// SIMATIC STEP 7 (V5.x) project PLC_PRV
// CPU: CPU 317-2 PN/DP
// station: Hardware
// station: SIMATIC 300 Station
// station: P_ADR_BUS
// program: S7 Program(6)

SYMBOL_TABLE
"RS485_chenal1"	DB 71	FB 72
"RS485_chanel2"	DB 72	FB 72
"RS485_chanel3"	DB 73	FB 72
"RS485_chanel4"	DB 74	FB 72
"KerVal1"	DB 101	FB 1
"ValGluchPerf"	DB 102	FB 1
"VidsmokVal"	DB 103	FB 1
"CalcRPM_Setka"	DB 104	FB 1
"CalcRPM_Gauch"	DB 105	FB 1
"CalcRPM_KerVal2"	DB 106	FB 1
"CalcRPM_JolVal"	DB 107	FB 1
"CalcRPM_Sushka1"	DB 108	FB 1
"CalcRPM_Sushka2"	DB 109	FB 1
"CalcRPM_Sushka3"	DB 110	FB 1
"CalcRPM_Sushka4"	DB 111	FB 1
"CalcRPM_KlejPresBNV1"	DB 112	FB 1
"CalcRPM_KlejPresBNV2"	DB 113	FB 1
"CalcRPM_KlejPresBNV3"	DB 114	FB 1
"CalcRPM_KlejPresBNV4"	DB 115	FB 1
"CalcRPM_KlejPresRuhVal"	DB 116	FB 1
"CalcRPM_KlejPresNeRuhVal"	DB 117	FB 1
"CalcRPM_Sushka5"	DB 118	FB 1
"CalcRPM_Sushka6"	DB 119	FB 1
"CalcRPM_Sushka7"	DB 120	FB 1
"CalcRPM_Kalandr"	DB 121	FB 1
"CalcRPM_Nakat"	DB 122	FB 1
"PaperVed1"	DB 123	FB 1
"PaperVedVal2"	DB 124	FB 1
"CalcRPM_PapVedVal3"	DB 125	FB 1
"CalcRPM_RozgonTambur"	DB 126	FB 1
"SpeedCalc_KombiPress"	DB 130	FB 2
"SpeedCalc_Sitka"	DB 131	FB 2
"CalcSpeed_Pres3"	DB 132	FB 2
"CalcSpeed_Sushka1"	DB 133	FB 2
"CalcSpeed_Sushka2"	DB 134	FB 2
"CalcSpeed_Sushka3"	DB 135	FB 2
"CalcSpeed_Sushka4"	DB 136	FB 2
"CalcSpeed_KlejPress"	DB 137	FB 2
"CalcSpeed_Sushka5"	DB 138	FB 2
"CalcSpeed_Sushka6"	DB 139	FB 2
"CalcSpeed_Sushka7"	DB 140	FB 2
"Signals_To_Nakat"	DB 201	DB 201
"PapVed1_Speed_Unit"	DB 203	FB 2
"PapVed2_Speed_Unit"	DB 204	FB 2
"PapVed3_Speed_Unit"	DB 205	FB 2
"Calc_RPM_Privod"	FB 1	FB 1	// Rozrahunok_RPM_privodiv
"Calc_Speed_Unit"	FB 2	FB 2	// Rozrahunok_shvidkosti_uzlov
"SEND"	FB 60	FB 60
"RECEIVE"	FB 61	FB 61
"RTU_MB_MASTER"	FB 72	FB 72
"RS485_1"	FC 1	FC 1	// RS485_1_Chanel
"RS485_2"	FC 2	FC 2	// RS485_2_chanel
"RS485_Runchanel3"	FC 3	FC 3
"RS485_RunChanel4"	FC 4	FC 4
"Speed_Calculation"	FC 10	FC 10	// Speed_Calculation
"RPM_Calculation"	FC 11	FC 11	// RPM_Calculation
"Speed_Intens"	FC 12	FC 12
"Calc_RPM_to_Hz"	FC 14	FC 14
"Calc_Zaprav_Speed"	FC 15	FC 15
"Check_AlarmPPS"	FC 30	FC 30
"UNSCALE"	FC 106	FC 106	// Unscaling Values
"SER_CFG"	FC 216	FC 216
"Kn_Zap_vidsm_val"	I 0.0	BOOL
"Vidsm_val_kontr_vkl"	I 0.2	BOOL
"Vidsm_val_kontR_blok"	I 0.4	BOOL
"Jolob_val_kont_kn_zapob"	I 0.5	BOOL
"Jolob_val_kont_vkl"	I 0.7	BOOL
"Jolob_val_kont_blok"	I 1.0	BOOL
"Keram_val1_kont_kn_zapob"	I 1.1	BOOL
"Keram_val1_kont_vkl"	I 1.3	BOOL
"Keram_val_1_kont_blok"	I 1.5	BOOL
"Ker_val2_konT_blok"	I 2.1	BOOL
"Ker_val_2_kont_kn_zapob"	I 2.4	BOOL
"Ker_val_2_kont_vkl"	I 2.6	BOOL
"Gluh_perf_kontr_kn_zapob"	I 3.0	BOOL
"Kalandr_kontrol_kn_zap"	I 9.0	BOOL
"Kalandr_kont_vkl"	I 9.2	BOOL
"Kalandr_kont_blokuvan"	I 9.4	BOOL
"Rozg_Tamb_Kn_Zap"	I 9.5	BOOL
"Rozg_Tamb_Kont_Vkl"	I 9.7	BOOL
"Rozg_Tamb_Kont_blok"	I 10.0	BOOL
"Nakat_kontrol_kn_zapob"	I 10.1	BOOL
"Nakat_kontrol_vkl"	I 10.3	BOOL
"Nakat_kontrol_blok"	I 10.5	BOOL
"MST_Zab_Zap_pres1_2_pik"	I 12.3	BOOL
"Z_MST_ZAB_zap_3_presu"	I 12.5	BOOL
"rez"	I 12.6	BOOL
"En_SitkVrusi"	M 20.0	BOOL	// Імітація сигналу на SCADA
"En_KombPresVroboti"	M 20.2	BOOL	// Імітація сигналу на SCADA
"Suska3_cor-"	M 20.3	BOOL
"En_Pres3Vroboti"	M 20.4	BOOL	// Імітація сигналу на SCADA
"Suska3_Pidtagnut"	M 20.5	BOOL
"Pusk_3pres"	M 20.6	BOOL	// Включити 3й прес HMI
"SitkaGaush_pusk"	M 20.7	BOOL	// Включити Сітка + гауч HMI_51
"Serv_mode_Sitka_Gauch"	M 21.1	BOOL
"Serv_mode_Kombi_Pres"	M 21.2	BOOL
"Serv_mode_Pres_3"	M 21.3	BOOL
"Serv_mode_Suska1"	M 21.6	BOOL
"Serv_mode_Suska2"	M 21.7	BOOL
"Serv_mode_Suska3"	M 22.0	BOOL
"Serv_mode_Suska4"	M 22.1	BOOL
"Serv_mode_BumNapr1"	M 22.2	BOOL
"Serv_mode_BumNapr2"	M 22.3	BOOL
"Serv_mode_BumNapr3"	M 22.4	BOOL
"Serv_mode_BumNapr4"	M 22.5	BOOL
"Serv_mode_RuhVal"	M 22.6	BOOL
"Serv_mode_NeruhVal"	M 22.7	BOOL
"Serv_mode_Suska5"	M 23.0	BOOL
"Serv_mode_Suska6"	M 23.1	BOOL
"Serv_mode_Suska7"	M 23.2	BOOL
"Serv_mode_PapVed3"	M 23.3	BOOL
"Serv_mode_Kalandr"	M 23.4	BOOL
"Serv_mode_Nakat"	M 23.5	BOOL
"Serv_mode_RozgTamb"	M 23.6	BOOL
"Suska4_cor+"	M 23.7	BOOL
"Suska4_cor-"	M 24.0	BOOL
"Suska4_Pidtagnut"	M 24.1	BOOL
"Suska5_cor+"	M 24.2	BOOL
"Suska5_cor-"	M 24.3	BOOL
"Suska5_Pidtagnut"	M 24.4	BOOL
"Suska6_cor+"	M 24.5	BOOL
"Suska6_cor-"	M 24.6	BOOL
"Suska6_Pidtagnut"	M 24.7	BOOL
"Suska7_cor+"	M 25.0	BOOL
"Suska7_cor-"	M 25.1	BOOL
"Suska7_Pidtagnut"	M 25.2	BOOL
"PaperVedVal2_Serv_mode"	M 25.3	BOOL
"PaperVedVal1_Serv_mode"	M 25.4	BOOL
"PaperVedVal1_Korec +"	M 25.5	BOOL
"PaperVedVal1_Korec -"	M 25.6	BOOL
"PaperVedVal2_Korec +"	M 25.7	BOOL
"PaperVedVal2_Korec -"	M 26.0	BOOL
"PaperVedVal3_Korec +"	M 26.1	BOOL
"PaperVedVal3_Korec -"	M 26.2	BOOL
"Gotovn_Kalandr"	M 800.0	BOOL
"Gotovn_Rozg_Tambur"	M 800.1	BOOL
"Gotovn_Nakat"	M 800.2	BOOL
"Dozv_Mash"	M 800.3	BOOL	// Загальний дозвіл машини
"PuskKerVal1"	M 999.0	BOOL
"Pusk_KombiPres"	M 999.1	BOOL	// Включити комбі прес HMI
"Pusk_Nakat"	M 1000.0	BOOL
"Pusk_Kalandr"	M 1001.0	BOOL
"Pusk_Suska7"	M 1002.0	BOOL
"Pusk_VidsmVal"	M 1003.0	BOOL
"Pusk_suska5"	M 1005.0	BOOL
"Pusk_Jolob_Val"	M 1010.0	BOOL
"PapVedVal_2_Pusk"	M 1022.0	BOOL
"Pusk_PapVed3"	M 1023.0	BOOL
"Pusk_Rozg_Tambur"	M 1024.0	BOOL
"Pusk_PapVedVal1"	M 1025.0	BOOL
"Pusk_KeramVal2"	M 1026.0	BOOL
"Pusk_ValGluhPerf"	M 1027.0	BOOL
"Pusk_Suska1"	M 1028.0	BOOL
"Pusk_suska6"	M 1029.0	BOOL
"Start_spov_val"	M 1029.1	BOOL
"pusk_sush2"	M 1029.2	BOOL
"Pusk_Sus_GR3"	M 1029.3	BOOL
"pusk_sgr4"	M 1029.4	BOOL
"pusk_gauc"	M 1029.5	BOOL
"doz_sgr4"	M 1029.6	BOOL
"sgr4_rst"	M 1029.7	BOOL
"En_dozv_Sus3"	M 1030.0	BOOL
"Rst_sus3"	M 1030.1	BOOL
"doz_sus2"	M 1030.2	BOOL
"rst_sgr2"	M 1030.3	BOOL
"Dozv_Sitka"	M 1030.4	BOOL
"rst_spvr"	M 1030.5	BOOL
"doz_gauch"	M 1030.6	BOOL
"rst_gauc"	M 1030.7	BOOL
"Dozv_kl_pr1"	M 1031.0	BOOL
"Pusk_Kl_pr2"	M 1031.2	BOOL
"Бум_напр_вал3_дозв_кн"	M 1031.6	BOOL
"Бум_напр_вал3_напр_кн"	M 1031.7	BOOL
"Pusk_BumNap3"	M 1032.0	BOOL
"Pusk_BumNap4"	M 1032.3	BOOL
"Pusk_PodvVal"	M 1032.6	BOOL
"Pusk_NepodvVal"	M 1033.1	BOOL
"Pres3_dod_svidk"	M 1508.6	BOOL
"Pres3_vidn_svidk"	M 1508.7	BOOL
"Pres3_Pidtygnut"	M 1509.0	BOOL
"Suska1_cor+"	M 1509.1	BOOL
"Suska1_cor-"	M 1509.2	BOOL
"Suska1_Pidtagnut"	M 1509.3	BOOL
"Suska2_cor+"	M 1509.4	BOOL
"Suska2_cor-"	M 1509.5	BOOL
"Suska2_Pidtagnut"	M 1509.6	BOOL
"Suska3_cor+"	M 1509.7	BOOL
"RS485_1_StartPaket"	M 1510.0	BOOL
"RS485_1_OK"	M 1510.1	BOOL
"RS485_1_ERR"	M 1510.2	BOOL
"RS485_1_Next"	M 1510.3	BOOL
"RS485_1_StopObmin"	M 1510.4	BOOL
"RS485_2_StartPaket"	M 1511.0	BOOL
"RS485_2_OK"	M 1511.1	BOOL
"RS485_2_ERR"	M 1511.2	BOOL
"RS485_2_Next"	M 1511.3	BOOL
"RS485_2_StopObmin"	M 1511.4	BOOL
"RS485_3_StartPaket"	M 1512.0	BOOL
"RS485_3_OK"	M 1512.1	BOOL
"RS485_3_ERR"	M 1512.2	BOOL
"RS485_3_Next"	M 1512.3	BOOL
"RS485_3_StopObmin"	M 1512.4	BOOL
"RS485_4_StartPaket"	M 1513.0	BOOL
"RS485_4_OK"	M 1513.1	BOOL
"RS485_4_ERR"	M 1513.2	BOOL
"RS485_4_Next"	M 1513.3	BOOL
"RS485_4_StopObmin"	M 1513.4	BOOL
"RS485_5_StartPaket"	M 1514.0	BOOL
"RS485_5_OK"	M 1514.1	BOOL
"RS485_5_ERR"	M 1514.2	BOOL
"RS485_5_Next"	M 1514.3	BOOL
"RS485_5_StopObmin"	M 1514.4	BOOL
"Speed_Mash"	MD 2000	DINT
"KerVal1_Dia"	MD 2008	DINT
"KerVal1_Kred"	MD 2012	DINT
"KerVal1_NNom"	MD 2016	DINT
"KerVal1_N0"	MD 2020	DINT
"KerVal1_RPMNom"	MD 2024	DINT
"KerVal2_Dia"	MD 2032	DINT
"KerVal2_Kred"	MD 2036	DINT
"KerVal2_NNom"	MD 2040	DINT
"KerVal2_N0"	MD 2044	DINT
"KerVal2_RPMNom"	MD 2048	DINT
"ValGluhPerf_Dia"	MD 2056	DINT
"ValGluhPerf_Kred"	MD 2060	DINT
"ValGluhPerf_Nnom"	MD 2064	DINT
"ValGluhPerf_N0"	MD 2068	DINT
"ValGluhPerf_RPMnom"	MD 2072	DINT
"Sushka1_Dia"	MD 2080	DINT
"Sushka1_Kred"	MD 2084	DINT
"Sushka1_NNom"	MD 2088	DINT
"Sushka1_N0"	MD 2092	DINT
"Sushka1_RPMNom"	MD 2096	DINT
"Sushka5_Dia"	MD 2104	DINT
"Sushka5_Kred"	MD 2108	DINT
"Sushka5_NNom"	MD 2112	DINT
"Sushka5_N0"	MD 2116	DINT
"Sushka5_RPMNom"	MD 2120	DINT
"Sushka6_Dia"	MD 2128	DINT
"Sushka6_Kred"	MD 2132	DINT
"Sushka6_NNom"	MD 2136	DINT
"Sushka6_N0"	MD 2140	DINT
"Sushka6_RPMNom"	MD 2144	DINT
"Sushka7_Dia"	MD 2152	DINT
"Sushka7_Kred"	MD 2156	DINT
"Sushka7_NNom"	MD 2160	DINT
"Sushka7_N0"	MD 2164	DINT
"Sushka7_RPMNom"	MD 2168	DINT
"Kalandr_Dia"	MD 2176	DINT
"Kalandr_Kred"	MD 2180	DINT
"Kalandr_NNom"	MD 2184	DINT
"Kalandr_N0"	MD 2188	DINT
"Kalandr_RPMNom"	MD 2192	DINT
"Nakat_Dia"	MD 2200	DINT
"Nakat_Kred"	MD 2204	DINT
"Nakat_NNom"	MD 2208	DINT
"Nakat_N0"	MD 2212	DINT
"Nakat_RPMNom"	MD 2216	DINT
"VidsmokVal_Dia"	MD 2224	DINT
"VidsmokVal_Kred"	MD 2228	DINT
"VidsmokVal_NNom"	MD 2232	DINT
"VidsmokVal_N0"	MD 2236	DINT
"VidsmokVal_RPMNom"	MD 2240	DINT
"JolVal_Dia"	MD 2248	DINT
"JolVal_Kred"	MD 2252	DINT
"JolVal_NNom"	MD 2256	DINT
"JolVal_N0"	MD 2260	DINT
"JolVal_RPMNom"	MD 2264	DINT
"PAPER_VED_1_KOEF_VIDHILU"	MD 2268	REAL
"PAPER_VED_1_D_vala"	MD 2272	DINT
"PAPER_VED_1_KOEF_REDUC"	MD 2276	DINT
"PAPER_VED_1_N_N0MIN"	MD 2280	DINT
"PAPER_VED_1_N_0"	MD 2284	DINT
"PAPER_VED_1_NOMIN_OBERT"	MD 2288	DINT
"PAPER_VED_2_KOEF_VIDHILU"	MD 2292	REAL
"PAPER_VED_2_D_vala"	MD 2296	DINT
"PAPER_VED_2_KOEF_REDUC"	MD 2300	DINT
"PAPER_VED_2_N_N0MIN"	MD 2304	DINT
"PAPER_VED_2_N_0"	MD 2308	DINT
"PAPER_VED_2_NOMIN_OBERT"	MD 2312	DINT
"PAPER_VED_3_KOEF_VIDHILU"	MD 2316	REAL
"PapVedVal3_Dia"	MD 2320	DINT
"PapVedVal3_Kred"	MD 2324	DINT
"PapVedVal3_NNom"	MD 2328	DINT
"PapVedVal3_N0"	MD 2332	DINT
"PapVedVal3_RPMNom"	MD 2336	DINT
"RozgonTambur_Dia"	MD 2344	DINT
"RozgonTambur_Kred"	MD 2348	DINT
"RozgonTambur_NNom"	MD 2352	DINT
"RozgonTambur_N0"	MD 2356	DINT
"RozgonTambur_RPMNom"	MD 2360	DINT
"Gauch_Dia"	MD 2368	DINT
"Gauch_Kred"	MD 2372	DINT
"Gauch_NNom"	MD 2376	DINT
"Gauch_N0"	MD 2380	DINT
"Gauch_RPMNom"	MD 2384	DINT
"Setka_Dia"	MD 2392	DINT
"Setka_Kred"	MD 2396	DINT
"Setka_NNom"	MD 2400	DINT
"Setka_N0"	MD 2404	DINT
"Setka_RPMNom"	MD 2408	DINT
"Sushka2_Dia"	MD 2416	DINT
"Sushka2_Kred"	MD 2420	DINT
"Sushka2_NNom"	MD 2424	DINT
"Sushka2_N0"	MD 2428	DINT
"Sushka2_RPMNom"	MD 2432	DINT
"Sushka3_Dia"	MD 2440	DINT
"Sushka3_Kred"	MD 2444	DINT
"Sushka3_NNom"	MD 2448	DINT
"Sushka3_N0"	MD 2452	DINT
"Sushka3_RPMNom"	MD 2456	DINT
"Sushka4_Dia"	MD 2464	DINT
"Sushka4_Kred"	MD 2468	DINT
"Sushka4_NNom"	MD 2472	DINT
"Sushka4_N0"	MD 2476	DINT
"Sushka4_RPMNom"	MD 2480	DINT
"KlejPresBumNap1_Dia"	MD 2488	DINT
"KlejPresBumNap1_Kred"	MD 2492	DINT
"KlejPresBumNap1_NNom"	MD 2496	DINT
"KlejPresBumNap1_N0"	MD 2500	DINT
"KlejPresBumNap1_RPMNom"	MD 2504	DINT
"KlejPresBumNap2_Dia"	MD 2512	DINT
"KlejPresBumNap2_Kred"	MD 2516	DINT
"KlejPresBumNap2_NNom"	MD 2520	DINT
"KlejPresBumNap2_N0"	MD 2524	DINT
"KlejPresBumNap2_RPMNom"	MD 2528	DINT
"KlejPresBumNap3_Dia"	MD 2536	DINT
"KlejPresBumNap3_Kred"	MD 2540	DINT
"KlejPresBumNap3_NNom"	MD 2544	DINT
"KlejPresBumNap3_N0"	MD 2548	DINT
"KlejPresBumNap3_RPMNom"	MD 2552	DINT
"KlejPresBumNap4_Dia"	MD 2560	DINT
"KlejPresBumNap4_Kred"	MD 2564	DINT
"KlejPresBumNap4_NNom"	MD 2568	DINT
"KlejPresBumNap4_N0"	MD 2572	DINT
"KlejPresBumNap4_RPMNom"	MD 2576	DINT
"KlejPresRuhVal_Dia"	MD 2584	DINT
"KlejPresRuhVal_Kred"	MD 2588	DINT
"KlejPresRuhVal_NNom"	MD 2592	DINT
"KlejPresRuhVal_N0"	MD 2596	DINT
"KlejPresRuhVal_RPMNom"	MD 2600	DINT
"KlejPresNeRuhVal_Dia"	MD 2608	DINT
"KlejPresNeRuhVal_Kred"	MD 2612	DINT
"KlejPresNeRuhVal_NNom"	MD 2616	DINT
"KlejPresNeRuhVal_N0"	MD 2620	DINT
"KlejPresNeRuhVal_RPMNom"	MD 2624	DINT
"Setka_Correction"	MD 2628	REAL
"KombiPress_Correction"	MD 2632	REAL
"Press3_Correction"	MD 2636	REAL
"Suchka1_Correction"	MD 2640	REAL
"Suchka2_Correction"	MD 2644	REAL
"Suchka3_Correction"	MD 2648	REAL
"Suchka4_Correction"	MD 2652	REAL
"Suchka5_Correction"	MD 2656	REAL
"Suchka6_Correction"	MD 2660	REAL
"Suchka7_Correction"	MD 2664	REAL
"KerVal1_RefOut"	MD 3000	DINT
"KerVal1_SpeedD"	MD 3004	DWORD
"KerVal2_RefOut"	MD 3008	DINT
"KerVal2_SpeedD"	MD 3012	DWORD
"ValGluhPerf_RefOut"	MD 3016	DINT
"ValGluhPerf_SpeedD"	MD 3020	DWORD
"Sushka1_RefOut"	MD 3024	DINT
"Sushka1_SpeedD"	MD 3028	DWORD
"Sushka5_RefOut"	MD 3032	DINT
"Sushka5_SpeedD"	MD 3036	DWORD
"Sushka6_RefOut"	MD 3040	DINT
"Sushka6_SpeedD"	MD 3044	DWORD
"Sushka7_RefOut"	MD 3048	DINT
"Sushka7_SpeedD"	MD 3052	DWORD
"Kalandr_RefOut"	MD 3056	DINT
"Kalandr_SpeedD"	MD 3060	DWORD
"Nakat_RefOut"	MD 3064	DINT
"Nakat_SpeedD"	MD 3068	DWORD
"VidsmokVal_RefOut"	MD 3072	DINT
"VidsmokVal_SpeedD"	MD 3076	DWORD
"JolVal_RefOut"	MD 3080	DINT
"JolVal_SpeedD"	MD 3084	DWORD
"PAPER_VED_1_To_AO_Cont"	MD 3088	DINT
"PAPER_VED_1_Spped_drive"	MD 3092	DWORD
"PAPER_VED_2_To_AO_Cont"	MD 3096	DINT
"PAPER_VED_2_Spped_drive"	MD 3100	DWORD
"PapVedVal3_RefOut"	MD 3104	DINT
"PapVedVal3_SpeedD"	MD 3108	DWORD
"RozgonTambur_RefOut"	MD 3112	DINT
"RozgonTambur_SpeedD"	MD 3116	DWORD
"Gauch_RefOut"	MD 3120	DINT
"Gauch_SpeedD"	MD 3124	DWORD
"Setka_RefOut"	MD 3128	DINT
"Setka_SpeedD"	MD 3132	DWORD
"Sushka2_RefOut"	MD 3136	DINT
"Sushka2_SpeedD"	MD 3140	DWORD
"Sushka3_RefOut"	MD 3144	DINT
"Sushka3_SpeedD"	MD 3148	DWORD
"Sushka4_RefOut"	MD 3152	DINT
"Sushka4_SpeedD"	MD 3156	DWORD
"Sushka1_RPM"	MD 3160	DINT
"Sushka5_RPM"	MD 3164	DINT
"KerVal1_RPM"	MD 3168	DINT
"KerVal2_RPM"	MD 3172	DINT
"ValGluhPerf_RPM"	MD 3176	DINT
"Sushka6_RPM"	MD 3180	DINT
"Sushka7_RPM"	MD 3184	DINT
"Kalandr_RPM"	MD 3188	DINT
"Nakat_RPM"	MD 3192	DINT
"VidsmokVal_RPM"	MD 3196	DINT
"JolVal_RPM"	MD 3200	DINT
"PAPER_VED_1_RPM"	MD 3204	DINT
"PAPER_VED_2_RPM"	MD 3208	DINT
"PapVedVal3_RPM"	MD 3212	DINT
"RozgonTambur_RPM"	MD 3216	DINT
"Gauch_RPM"	MD 3220	DINT
"Setka_RPM"	MD 3224	DINT
"Sushka2_RPM"	MD 3228	DINT
"Sushka3_RPM"	MD 3232	DINT
"Sushka4_RPM"	MD 3236	DINT
"KlejPresBumNap1_RefOut"	MD 3240	DINT
"KlejPresBumNap1_SpeedD"	MD 3244	DWORD
"KlejPresBumNap1_RPM"	MD 3248	DINT
"KlejPresBumNap2_RefOut"	MD 3252	DINT
"KlejPresBumNap2_SpeedD"	MD 3256	DWORD
"KlejPresBumNap2_RPM"	MD 3260	DINT
"KlejPresBumNap3_RefOut"	MD 3264	DINT
"KlejPresBumNap3_SpeedD"	MD 3268	DWORD
"KlejPresBumNap3_RPM"	MD 3272	DINT
"KlejPresRuhVal_RefOut"	MD 3276	DINT
"KlejPresRuhVal_SpeedD"	MD 3280	DWORD
"KlejPresRuhVal_RPM"	MD 3284	DINT
"KlejPresNeRuhVal_RefOut"	MD 3288	DINT
"KlejPresNeRuhVal_SpeedD"	MD 3292	DWORD
"KlejPresNeRuhVal_RPM"	MD 3296	DINT
"KlejPresBumNap4_RefOut"	MD 3300	DINT
"KlejPresBumNap4_SpeedD"	MD 3304	DWORD
"KlejPresBumNap4_RPM"	MD 3308	DINT
"Speed_Mash_Zad_R"	MD 4600	REAL
"Speed_Mash_Pot_R"	MD 4604	REAL
"Speed_KombiPressR"	MD 4608	REAL
"Speed_SetkaR"	MD 4612	REAL
"Speed_Pres3_R"	MD 4616	REAL
"Speed_Suchka1_R"	MD 4620	REAL
"Speed_Suchka2_R"	MD 4624	REAL
"Speed_Suchka3_R"	MD 4628	REAL
"Speed_Suchka4_R"	MD 4632	REAL
"Speed_KlajPress_R"	MD 4636	REAL
"Speed_Suchka5_R"	MD 4640	REAL
"Speed_Suchka6_R"	MD 4644	REAL
"Speed_Suchka7_R"	MD 4648	REAL
"Speed_Kalandr"	MD 4652	REAL
"Speed_Nakat"	MD 4656	REAL
"Speed_KombiPress_Zapr"	MD 4684	REAL
"Speed_Setka_gauch_Zapr"	MD 4688	REAL
"Speed_Pres3_Zapr"	MD 4692	REAL
"Speed_Suchka1_Zapr"	MD 4696	REAL
"Speed_Suchka2_Zapr"	MD 4700	REAL
"Speed_Suchka 3_Zapr"	MD 4704	REAL
"Speed_Suchka 4_Zapr"	MD 4708	REAL
"Speed_Suchka 5_Zapr"	MD 4712	REAL
"Speed_Suchka 6_Zapr"	MD 4716	REAL
"Speed_Suchka 7_Zapr"	MD 4720	REAL
"Speed_Kalandr_Zapr"	MD 4724	REAL
"Speed_Nakat_Zapr"	MD 4728	REAL
"Speed_BumNaprVal1_Zapr"	MD 4732	REAL
"Speed_BumNaprVal2_Zapr"	MD 4736	REAL
"Speed_BumNaprVal3_Zapr"	MD 4740	REAL
"Speed_BumNaprVal4_Zapr"	MD 4744	REAL
"Speed_RuhVal_Zapr"	MD 4748	REAL
"Speed_NeRuhVal_Zapr"	MD 4752	REAL
"Speed_PaperVed2"	MD 4756	REAL
"Speed_PaperVed3_Zapr"	MD 4760	REAL
"Speed_PaperVed1_Zapr"	MD 4764	REAL
"Speed_RozgTamb_Zapr"	MD 4768	REAL
"Current_Speed_Sitka"	MD 4772	REAL
"Current_Speed_Kombi_pres"	MD 4776	REAL
"Current_Speed_Press3"	MD 4780	REAL
"Current_Speed_Sushka 1"	MD 4784	REAL
"Curr_Speed_GauchVal"	MD 4788	REAL
"Curr_Speed_KerVal2"	MD 4792	REAL
"Curr_Speed_JolbVal"	MD 4796	REAL
"Curr_Speed_VidsmVal"	MD 4800	REAL
"Curr_Speed_GluhPerf"	MD 4804	REAL
"Curr_Speed_Suska1"	MD 4812	REAL
"Curr_Speed_Suska2"	MD 4816	REAL
"Curr_Speed_Suska3"	MD 4820	REAL
"Curr_Speed_Suska4"	MD 4824	REAL
"Curr_Speed_BumNap1"	MD 4828	REAL
"Curr_Speed_BumNap2"	MD 4832	REAL
"Curr_Speed_BumNap3"	MD 4836	REAL
"Curr_Speed_BumNap4"	MD 4840	REAL
"Curr_Speed_RuhVal"	MD 4844	REAL
"Curr_Speed_NeRuhVal"	MD 4848	REAL
"Curr_Speed_Suska5"	MD 4852	REAL
"Curr_Speed_Suska6"	MD 4856	REAL
"Curr_Speed_Suska7"	MD 4860	REAL
"Curr_Speed_PapVed3"	MD 4864	REAL
"Curr_Speed_Kalandr"	MD 4868	REAL
"Curr_Speed_Nakat"	MD 4872	REAL
"Curr_Speed_RozgTambur"	MD 4876	REAL
"Curr_Speed_PapVed2"	MD 4880	REAL
"Curr_Speed_PapVed1"	MD 4884	REAL
"Speed_PapVed1"	MD 4888	REAL
"Speed_PapVed2"	MD 4892	REAL
"Speed_PapVed3"	MD 4896	REAL
"RS485_1_CodErr"	MW 1515	WORD
"RS485_2_CodErr"	MW 1517	WORD
"RS485_3_CodErr"	MW 1519	WORD
"RS485_4_CodErr"	MW 1521	WORD
"RS485_5_CodErr"	MW 1523	WORD
"RS485_1_Count"	MW 1525	INT
"RS485_2_Count"	MW 1527	INT
"RS485_3_Count"	MW 1529	INT
"RS485_4_Count"	MW 1531	INT
"RS485_5_Count"	MW 1533	INT
"Keram_val_1_CurSpeed"	MW 4000	WORD
"Keram_val_1_Moment"	MW 4002	WORD
"Keram_val_1_Current"	MW 4004	WORD
"Keram_val_1_Udvg"	MW 4006	WORD
"Keram_val_1_Izbudj"	MW 4008	WORD
"Keram_val_1_Uzbudj"	MW 4010	WORD
"Keram_val_2_CurSpeed"	MW 4020	WORD
"Keram_val_2_Moment"	MW 4022	WORD
"Keram_val_2_Current"	MW 4024	WORD
"Keram_val_2_Udvg"	MW 4026	WORD
"Keram_val_2_Izbudj"	MW 4028	WORD
"Keram_val_2_Uzbudj"	MW 4030	WORD
"Val_z_gluh_perf_CurSpeed"	MW 4040	WORD
"Val_z_gluh_perf_Moment"	MW 4042	WORD
"Val_z_gluh_perf_Current"	MW 4044	WORD
"Val_z_gluh_perf_Udvg"	MW 4046	WORD
"Val_z_gluh_perf_Izbudj"	MW 4048	WORD
"Val_z_gluh_perf_Uzbudj"	MW 4050	WORD
"Suska_1_CurSpeed"	MW 4060	WORD
"Suska_1_Moment"	MW 4062	WORD
"Suska_1_Current"	MW 4064	WORD
"Suska_1_Udvg"	MW 4066	WORD
"Suska_1_Izbudj"	MW 4068	WORD
"Suska_1_Uzbudj"	MW 4070	WORD
"Suska_6_CurSpeed"	MW 4100	WORD
"Suska_6_Moment"	MW 4102	WORD
"Suska_6_Current"	MW 4104	WORD
"Suska_6_Udvg"	MW 4106	WORD
"Suska_6_Izbudj"	MW 4108	WORD
"Suska_6_Uzbudj"	MW 4110	WORD
"Suska_7_CurSpeed"	MW 4120	WORD
"Suska_7_Moment"	MW 4122	WORD
"Suska_7_Current"	MW 4124	WORD
"Suska_7_Udvg"	MW 4126	WORD
"Suska_7_Izbudj"	MW 4128	WORD
"Suska_7_Uzbudj"	MW 4130	WORD
"Kalandr_CurSpeed"	MW 4140	WORD
"Kalandr_Moment"	MW 4142	WORD
"Kalandr_Current"	MW 4144	WORD
"Kalandr_Udvg"	MW 4146	WORD
"Kalandr_Izbudj"	MW 4148	WORD
"Kalandr_Uzbudj"	MW 4150	WORD
"Nakat_CurSpeed"	MW 4160	WORD
"Nakat_Moment"	MW 4162	WORD
"Nakat_Current"	MW 4164	WORD
"Nakat_Udvg"	MW 4166	WORD
"Nakat_Izbudj"	MW 4168	WORD
"Nakat_Uzbudj"	MW 4170	WORD
"VidsmokVal_CurSpeed"	MW 4180	WORD
"VidsmokVal_Moment"	MW 4182	WORD
"VidsmokVal_Current"	MW 4184	WORD
"VidsmokVal_Udvg"	MW 4186	WORD
"VidsmokVal_Izbudj"	MW 4188	WORD
"VidsmokVal_Uzbudj"	MW 4190	WORD
"Suska_5_CurSpeed"	MW 4200	WORD
"Suska_5_Moment"	MW 4202	WORD
"Suska_5_Current"	MW 4204	WORD
"Suska_5_Udvg"	MW 4206	WORD
"Suska_5_Izbudj"	MW 4208	WORD
"Suska_5_Uzbudj"	MW 4210	WORD
"RozgonTambur_CurSpeed"	MW 4220	WORD
"RozgonTambur_Moment"	MW 4222	WORD
"RozgonTambur_Current"	MW 4224	WORD
"RozgonTambur_Udvg"	MW 4226	WORD
"RozgonTambur_Izbudj"	MW 4228	WORD
"RozgonTambur_Uzbudj"	MW 4230	WORD
"PapVedVal1_CurSpeed"	MW 4240	WORD
"PapVedVal1_Moment"	MW 4242	WORD
"PapVedVal1_Current"	MW 4244	WORD
"PapVedVal1_Udvg"	MW 4246	WORD
"PapVedVal1_Izbudj"	MW 4248	WORD
"PapVedVal1_Uzbudj"	MW 4250	WORD
"PapVedVal2_CurSpeed"	MW 4260	WORD
"PapVedVal2_Moment"	MW 4262	WORD
"PapVedVal2_Current"	MW 4264	WORD
"PapVedVal2_Udvg"	MW 4266	WORD
"PapVedVal2_Izbudj"	MW 4268	WORD
"PapVedVal2_Uzbudj"	MW 4270	WORD
"PapVedVal3_CurSpeed"	MW 4280	WORD
"PapVedVal3_Moment"	MW 4282	WORD
"PapVedVal3_Current"	MW 4284	WORD
"PapVedVal3_Udvg"	MW 4286	WORD
"PapVedVal3_Izbudj"	MW 4288	WORD
"PapVedVal3_Uzbudj"	MW 4290	WORD
"PapNapVal1_CurSpeed"	MW 4300	WORD
"PapNapVal1_Moment"	MW 4302	WORD
"PapNapVal1_Current"	MW 4304	WORD
"PapNapVal1_Udvg"	MW 4306	WORD
"State_Of_PapVedVal1"	MW 4308	WORD
"JolobVal_CurSpeed"	MW 4420	WORD
"JolobVal_Moment"	MW 4422	WORD
"JolobVal_Current"	MW 4424	WORD
"JolobVal_Udvg"	MW 4426	WORD
"JolobVal_Izbudj"	MW 4428	WORD
"JolobVal_Uzbudj"	MW 4430	WORD
"Speed_Hz_BumNapVal1"	MW 4660	WORD
"Speed_Hz_BumNapVal2"	MW 4662	WORD
"Speed_Hz_BumNapVal3"	MW 4664	WORD
"Speed_Hz_BumNapVal4"	MW 4666	WORD
"Speed_Hz_RuchVal"	MW 4668	WORD
"Speed_Hz_NeRuchVal"	MW 4670	WORD
"CodErr_KerVal1"	MW 5000	WORD
"CodErr_VidsmVal"	MW 5002	WORD
"CodErr_ValGluch"	MW 5004	WORD
"UK_Obm485_2"	MW 15004	WORD
"COMPLETE RESTART"	OB 100	OB 100	// Complete Restart
"VDSM_V"	PQW 272	INT
"KERAM_1"	PQW 274	INT
"JOLOBVAL"	PQW 276	INT
"KERAM_2"	PQW 278	INT	// Сигнал траолляля
"GLUH142"	PQW 280	INT
"PV2"	PQW 282	INT
"PV1"	PQW 284	INT
"SUH_G1"	PQW 286	INT
"SUH_G5"	PQW 288	INT
"SUH_G7"	PQW 290	INT
"SUH_G6"	PQW 292	INT
"VED_V3"	PQW 294	INT
"KALANDR"	PQW 296	INT
"NAKAT"	PQW 298	INT
"ROZ_TAMB"	PQW 300	INT
"Sitka_Pov_v_AO"	PQW 302	INT
"Gauch_AO"	PQW 304	INT
"Suska3_AO"	PQW 306	INT
"Suska2_AO"	PQW 308	INT
"Suska4_AO"	PQW 310	INT
"KL_PRES1_AO"	PQW 312	INT
"Pap_nap3_AO"	PQW 314	INT
"KL_PRES2_AO"	PQW 316	INT
"Pap_napr4_AO"	PQW 318	INT
"Podv_val_AO"	PQW 320	INT
"X7_AO2"	PQW 322	INT
"Nepod_val_AO"	PQW 324	INT
"hzhz2"	PQW 328	INT
"Run_VidsmVal"	Q 0.0	BOOL
"Run_ValGluhPerf"	Q 0.1	BOOL
"Run_JolobVal"	Q 0.2	BOOL
"Run_PapVedVal1"	Q 0.3	BOOL
"Run_KerVal1"	Q 0.4	BOOL
"PapVedVal_2_Run"	Q 0.5	BOOL
"Run_KeramVal2"	Q 0.6	BOOL
"Run_Suska1"	Q 0.7	BOOL
"Run_Suska5"	Q 1.0	BOOL
"Run_Kalandr"	Q 1.1	BOOL
"Run_Suska6"	Q 1.2	BOOL
"Run_Rozg_Tambur"	Q 1.3	BOOL
"Run_Suska7"	Q 1.4	BOOL
"Start_Nakat"	Q 1.5	BOOL
"Run_PapVed3"	Q 1.6	BOOL
"Sitka_dozvil"	Q 1.7	BOOL
"Sitka_reset_err"	Q 2.0	BOOL
"GauchVal_Run"	Q 2.1	BOOL
"Sitka_Run"	Q 2.2	BOOL
"Dozv_SUS2"	Q 2.3	BOOL
"Dozv_Gauch"	Q 2.4	BOOL
"Sus2_Reset_err"	Q 2.5	BOOL
"rst_Gauch"	Q 2.6	BOOL
"Run_Suska2"	Q 2.7	BOOL
"Dozvil_SUS3"	Q 3.0	BOOL
"Suska4_Reset_err"	Q 3.1	BOOL
"Suska3_Reset_err"	Q 3.2	BOOL
"Run_Suska4"	Q 3.3	BOOL
"Suska3_Run"	Q 3.4	BOOL
"Dozvil_KLEIL_PRES1"	Q 3.5	BOOL
"Dozvil_SUS4"	Q 3.6	BOOL
"Napr_kl_pr1"	Q 3.7	BOOL
"Start_KL_PR1"	Q 4.0	BOOL
"Змін_напр_бум_напр_вал3"	Q 4.1	BOOL
"Dozv_kl_pr2"	Q 4.2	BOOL
"Dozv_PapNap3"	Q 4.3	BOOL
"Napr_kl_pr2"	Q 4.4	BOOL
"Run_PapNap3"	Q 4.5	BOOL
"Start_kl_pr2"	Q 4.6	BOOL
"Dozv_pap_napr4"	Q 4.7	BOOL
"Napr_bum_napr4"	Q 5.0	BOOL
"Run_Podv_val"	Q 5.1	BOOL
"Run_bum_napr4"	Q 5.2	BOOL
"Dozvil_Nepod_Val"	Q 5.3	BOOL
"Dozv_Podv_val"	Q 5.4	BOOL
"Napr_Nepod_val"	Q 5.5	BOOL
"Napr_Podv_val"	Q 5.6	BOOL
"Run_Nepod_val"	Q 5.7	BOOL
"To_mst_Sitka_v_Rusi"	Q 6.0	BOOL
"xz"	Q 6.1	BOOL
"To_MST_Work_3x_presses"	Q 6.2	BOOL
"xxx"	Q 6.3	BOOL
"To_MST_Rob_3go_presu"	Q 6.4	BOOL
"z"	Q 7.0	BOOL
"Signal_MST1"	Q 7.1	BOOL
"Signal_MST2"	Q 7.2	BOOL
"Signal _mst3"	Q 7.3	BOOL
"TON"	SFB 4	SFB 4	// Generate an On Delay
"GET"	SFB 14	SFB 14	// Read Data From a Remote CPU
"DPRD_DAT"	SFC 14	SFC 14	// Read Consistent Data of a Standard DP Slave
"DPWR_DAT"	SFC 15	SFC 15	// Write Consistent Data to a Standard DP Slave
"BLKMOV"	SFC 20	SFC 20	// Copy Variables
"FILL"	SFC 21	SFC 21	// Initialize a Memory Area
"doz_rst"	T 0	TIMER
"RS485_1_Timer"	T 11	TIMER
"RS485_2_Timer"	T 12	TIMER
"RS485_3_Timer"	T 13	TIMER
"RS485_4_Timer"	T 14	TIMER
"RS485_5_Timer"	T 15	TIMER
END_SYMBOL_TABLE

FUNCTION_BLOCK "Calc_RPM_Privod"	// FB 1
VERSION : 0.1
VAR_INPUT
  S_PRIVOD_R : REAL ;
  D_VALA : DINT ;
  KOEF_RED : DINT ;
  N_NOMIN : DINT ;
  N_0 : DINT ;
  OBR_NOM : DINT ;
  Service_mode : BOOL ;
  Service_Speed : REAL ;
  Input_RPM : WORD ;
END_VAR
VAR_OUTPUT
  RESULT_N_ZAVD : DINT ;
  S_PRIVOD_D : DWORD ;
  RPM_DVIG : DINT ;
  Cur_Speed : REAL ;
END_VAR
VAR
  S_MASH_R : REAL ;
  KOEF_VIDHILU_R : REAL ;
  D_VALA_R : REAL ;
  KOEF_RED_R : REAL ;
  N_NOMIN_R : REAL ;
  N_0_R : REAL ;
  OBR_NOM_R : REAL ;
  TEMP_R : REAL ;
  TEMP_DINT : DINT ;
  KMUL : REAL ;
  N_VALA_R : REAL ;
  N_DVIG_R : REAL ;
  STAT0 : REAL ;
  N_MAX_R : REAL ;
  TEMP_2_R : REAL ;
  N_ZADANIE_R : REAL ;
  BIPOLAR : BOOL ;
  RET : WORD ;
  TEMP_RESULT : DINT ;
  TEMP_VAL_R : REAL ;
  TEMP_DVG_R : REAL ;
END_VAR
VAR_TEMP
  Calc_Speed : REAL ;
END_VAR
BEGIN
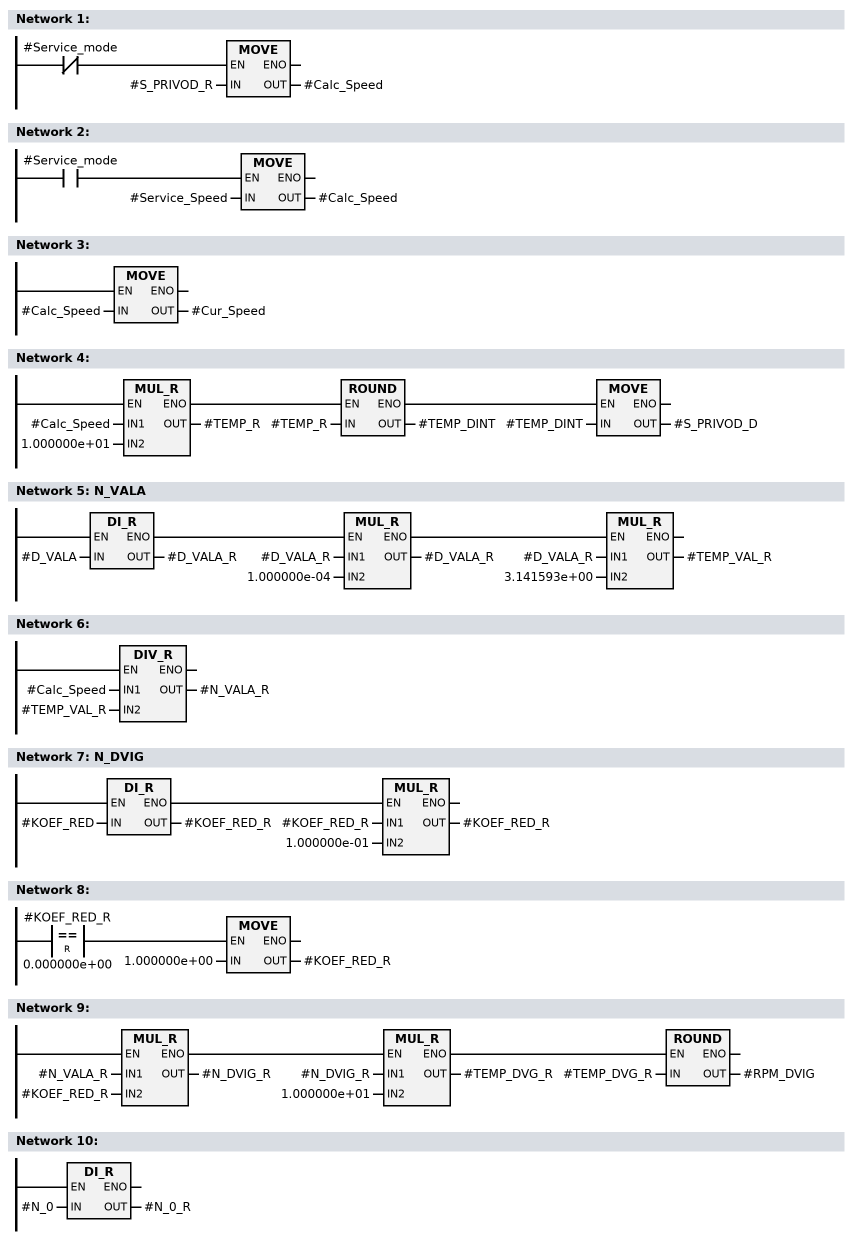
NETWORK
TITLE =
      AN    #Service_mode;
      JNB   _001;
      L     #S_PRIVOD_R;
      T     #Calc_Speed;
_001: NOP   0;
NETWORK
TITLE =
      A     #Service_mode;
      JNB   _002;
      L     #Service_Speed;
      T     #Calc_Speed;
_002: NOP   0;
NETWORK
TITLE =
      L     #Calc_Speed;
      T     #Cur_Speed;
      NOP   0;
NETWORK
TITLE =
      A(;
      A(;
      L     #Calc_Speed;
      L     1.000000e+01;
      *R;
      T     #TEMP_R;
      AN    OV;
      SAVE;
      CLR;
      A     BR;
      );
      JNB   _003;
      L     #TEMP_R;
      RND;
      T     #TEMP_DINT;
      AN    OV;
      SAVE;
      CLR;
_003: A     BR;
      );
      JNB   _004;
      L     #TEMP_DINT;
      T     #S_PRIVOD_D;
_004: NOP   0;
NETWORK
TITLE = N_VALA
      A(;
      A(;
      L     #D_VALA;
      DTR;
      T     #D_VALA_R;
      SET;
      SAVE;
      CLR;
      A     BR;
      );
      JNB   _005;
      L     #D_VALA_R;
      L     1.000000e-04;
      *R;
      T     #D_VALA_R;
      AN    OV;
      SAVE;
      CLR;
_005: A     BR;
      );
      JNB   _006;
      L     #D_VALA_R;
      L     3.141593e+00;
      *R;
      T     #TEMP_VAL_R;
_006: NOP   0;
NETWORK
TITLE =
      L     #Calc_Speed;
      L     #TEMP_VAL_R;
      /R;
      T     #N_VALA_R;
      NOP   0;
NETWORK
TITLE = N_DVIG
      A(;
      L     #KOEF_RED;
      DTR;
      T     #KOEF_RED_R;
      SET;
      SAVE;
      CLR;
      A     BR;
      );
      JNB   _007;
      L     #KOEF_RED_R;
      L     1.000000e-01;
      *R;
      T     #KOEF_RED_R;
_007: NOP   0;
NETWORK
TITLE =
      A(;
      L     #KOEF_RED_R;
      L     0.000000e+00;
      ==R;
      );
      JNB   _008;
      L     1.000000e+00;
      T     #KOEF_RED_R;
_008: NOP   0;
NETWORK
TITLE =
      A(;
      A(;
      L     #N_VALA_R;
      L     #KOEF_RED_R;
      *R;
      T     #N_DVIG_R;
      AN    OV;
      SAVE;
      CLR;
      A     BR;
      );
      JNB   _009;
      L     #N_DVIG_R;
      L     1.000000e+01;
      *R;
      T     #TEMP_DVG_R;
      AN    OV;
      SAVE;
      CLR;
_009: A     BR;
      );
      JNB   _00a;
      L     #TEMP_DVG_R;
      RND;
      T     #RPM_DVIG;
_00a: NOP   0;
NETWORK
TITLE =
      L     #N_0;
      DTR;
      T     #N_0_R;
      NOP   0;
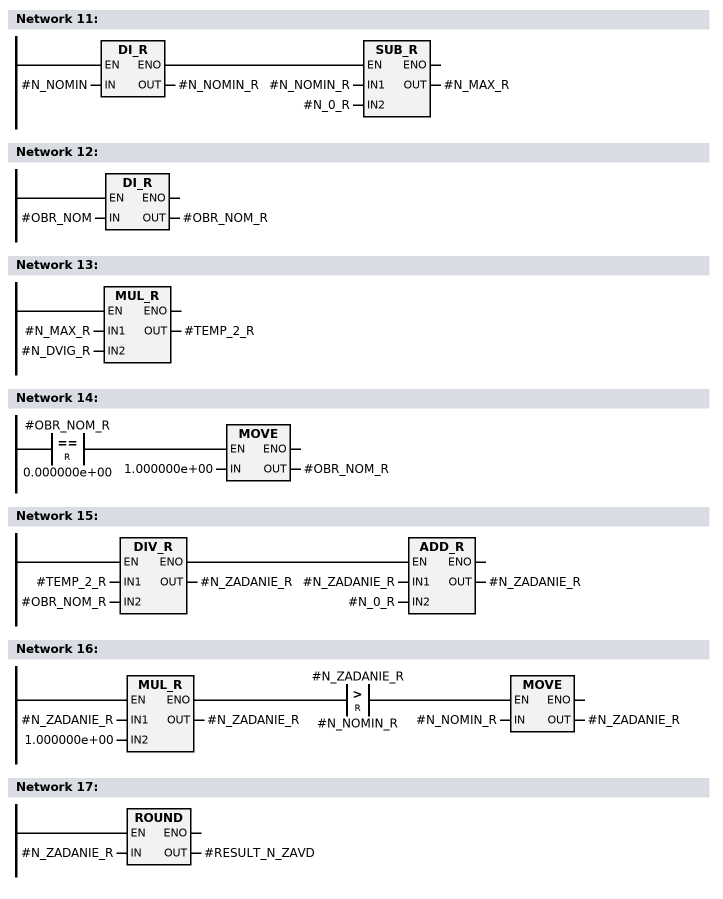
NETWORK
TITLE =
      A(;
      L     #N_NOMIN;
      DTR;
      T     #N_NOMIN_R;
      SET;
      SAVE;
      CLR;
      A     BR;
      );
      JNB   _00b;
      L     #N_NOMIN_R;
      L     #N_0_R;
      -R;
      T     #N_MAX_R;
_00b: NOP   0;
NETWORK
TITLE =
      L     #OBR_NOM;
      DTR;
      T     #OBR_NOM_R;
      NOP   0;
NETWORK
TITLE =
      L     #N_MAX_R;
      L     #N_DVIG_R;
      *R;
      T     #TEMP_2_R;
      NOP   0;
NETWORK
TITLE =
      A(;
      L     #OBR_NOM_R;
      L     0.000000e+00;
      ==R;
      );
      JNB   _00c;
      L     1.000000e+00;
      T     #OBR_NOM_R;
_00c: NOP   0;
NETWORK
TITLE =
      A(;
      L     #TEMP_2_R;
      L     #OBR_NOM_R;
      /R;
      T     #N_ZADANIE_R;
      AN    OV;
      SAVE;
      CLR;
      A     BR;
      );
      JNB   _00d;
      L     #N_ZADANIE_R;
      L     #N_0_R;
      +R;
      T     #N_ZADANIE_R;
_00d: NOP   0;
NETWORK
TITLE =
      A(;
      L     #N_ZADANIE_R;
      L     1.000000e+00;
      *R;
      T     #N_ZADANIE_R;
      AN    OV;
      SAVE;
      CLR;
      A     BR;
      );
      A(;
      L     #N_ZADANIE_R;
      L     #N_NOMIN_R;
      >R;
      );
      JNB   _00e;
      L     #N_NOMIN_R;
      T     #N_ZADANIE_R;
_00e: NOP   0;
NETWORK
TITLE =
      L     #N_ZADANIE_R;
      RND;
      T     #RESULT_N_ZAVD;
      NOP   0;
END_FUNCTION_BLOCK

FUNCTION_BLOCK "Calc_Speed_Unit"	// FB 2
VERSION : 0.1
VAR_INPUT
  S_Privoda_pochatkova : REAL ;
  Dodat_svidkist : BOOL ;
  Vidnyat_svidkist : BOOL ;
  Pidtyagnut : BOOL ;
  Percent_In : REAL ;
END_VAR
VAR_OUTPUT
  S_Privoda_rozrah : REAL ;
  Percent_Out : REAL ;
END_VAR
VAR
  TempPl : BOOL ;
  TempMn : BOOL ;
END_VAR
VAR_TEMP
  Percent : REAL ;
  PercentD : REAL ;
  Percent_Ras : REAL ;
  PercentR1 : REAL ;
  PercentR2 : REAL ;
END_VAR
BEGIN
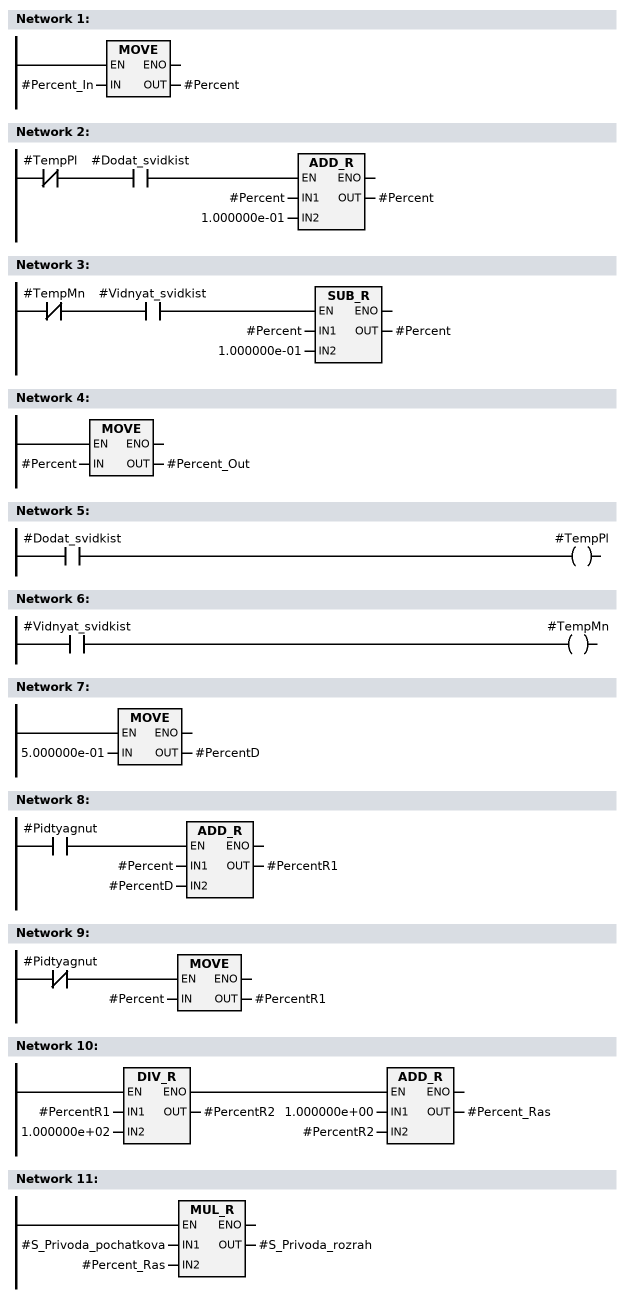
NETWORK
TITLE =
      L     #Percent_In;
      T     #Percent;
      NOP   0;
NETWORK
TITLE =
      AN    #TempPl;
      A     #Dodat_svidkist;
      JNB   _001;
      L     #Percent;
      L     1.000000e-01;
      +R;
      T     #Percent;
_001: NOP   0;
NETWORK
TITLE =
      AN    #TempMn;
      A     #Vidnyat_svidkist;
      JNB   _002;
      L     #Percent;
      L     1.000000e-01;
      -R;
      T     #Percent;
_002: NOP   0;
NETWORK
TITLE =
      L     #Percent;
      T     #Percent_Out;
      NOP   0;
NETWORK
TITLE =
      A     #Dodat_svidkist;
      =     #TempPl;
NETWORK
TITLE =
      A     #Vidnyat_svidkist;
      =     #TempMn;
NETWORK
TITLE =
      L     5.000000e-01;
      T     #PercentD;
      NOP   0;
NETWORK
TITLE =
      A     #Pidtyagnut;
      JNB   _003;
      L     #Percent;
      L     #PercentD;
      +R;
      T     #PercentR1;
_003: NOP   0;
NETWORK
TITLE =
      AN    #Pidtyagnut;
      JNB   _004;
      L     #Percent;
      T     #PercentR1;
_004: NOP   0;
NETWORK
TITLE =
      A(;
      L     #PercentR1;
      L     1.000000e+02;
      /R;
      T     #PercentR2;
      AN    OV;
      SAVE;
      CLR;
      A     BR;
      );
      JNB   _005;
      L     1.000000e+00;
      L     #PercentR2;
      +R;
      T     #Percent_Ras;
_005: NOP   0;
NETWORK
TITLE =
      L     #S_Privoda_pochatkova;
      L     #Percent_Ras;
      *R;
      T     #S_Privoda_rozrah;
      NOP   0;
END_FUNCTION_BLOCK

FUNCTION_BLOCK "SEND"	// FB 60
TITLE = SEND
//History:
//V1.0   erste Version
//V1.1   Sprungmarke T030 -> von #bFragCounter werden nur noch die untersten 3 Bit
//       in das Control-Wort geschrieben
//       Sprungmarke S050 --> Korrektur der Berechnung von wTemp1
//V1.2   Ьbergabe BLKMOV RetVal an Status
//       Reset auch bei fehlerhaften Eingangsparametern möglich
//       Ausgangsbits stehen nur für einen SPS-Zyklus an
//       Status 0x0517 und 0x070A hinzugefügt
//V1.3   neuer interner Status ERROR hinzugefügt
//V2.0   Prozessdatenzugriff auf SFC14/15 umgestellt
//V2.1   Längenkorrektur Destination-Pointer für Block-Move in NW8 beim Schreiben 
//       vom Header und Header/Trailer kombiniert
VERSION : 2.1
VAR_INPUT
  REQ : BOOL ;	//AuftragsanstoЯ bei positiver Flanke
  R : BOOL ;	//Synchron Reset auslösen
  LADDR : INT ;	//logische Basisadresse des CP - entspricht der Adresse aus der HW-Konfiguration
  DB_NO : INT ;	//Datenbausteinnummer - Nummer des Sende-DB (>0)
  DBB_NO : INT ;	//Datenbytenummer - Sendedaten ab Datenbyte
  LEN : INT ;	//Länge des zu sendenen Telegramms in Byte (>0 und <1025)
  IO_SIZE : WORD ;	//parametrierte IO Größe des Moduls
END_VAR
VAR_OUTPUT
  DONE : BOOL ;	//Auftrag fertig ohne Fehler, Daten gesendet, Parameter STATUS=00h
  ERROR : BOOL ;	//Auftrag fertig mit Fehler, Parameter STATUS enthält die Fehlerinformation
  STATUS : WORD ;	//Spezifikation des Fehlers bei ERROR=1
END_VAR
VAR_IN_OUT
  CONTROL : BYTE ;	//geteilter Speicher: Sendebaustein Bit 0..3, Empfangsbaustein Bit 4-7
END_VAR
VAR
  bIntStatus : BYTE ;	//interner Bausteinstatus
  bAcknowledge : BYTE ;	//Bit 4..7 des Eingangsbyte 0 als Quittung
  bFrag : BYTE ;	//Fragmentanzahl
  bFragCounter : BYTE ;	//Fragmentzähler
  xFpRequest : BOOL ;	//Hilfsbit zur Erkennung einer steigenden Flanke an REQ
  xFpReset : BOOL ;	//Hilfsbit zur Erkennung einer steigenden Flanke an R
  xResetDone : BOOL ;	//Fertigmeldung Synchron Reset (Statemachine Bit)
  iLenTrailer : INT ;	//Trailer Länge = Anzahl Nutzdaten im Trailer
  xResetBecauseAbort : BOOL ;	//Reset durch fallende Flanke an REQ ausgelöst
  xWait : BOOL ;	//warte nach fertigem Reset oder Auftrag mit Fehler auf FALS an EN_R und R
  wStatusMem : WORD ;	//temporärer Zwischenspeicher für STATUS Ausgang
  arInputData : ARRAY  [0 .. 59 ] OF BYTE ;
  arOutputData : ARRAY  [0 .. 59 ] OF BYTE ;
END_VAR
VAR_TEMP
  anyScr : ANY ;
  anyDst : ANY ;
  iRetval : INT ;
  wTemp1 : WORD ;
  wTemp2 : WORD ;
  dwTemp1 : DWORD ;
  dwTemp2 : DWORD ;
  wLaddr : WORD ;
END_VAR
BEGIN
NETWORK
TITLE = INIT
//
//Sprungmarken Definition:
//   Ixxx INIT
//   Rxxx SCHREIBE RESET
//   Sxxx START
//   Txxx SENDEN
//   Qxxx TLG QUITTUNG
//   Axxx ABSCHLIEЯEN
//   Exxx ENDE
//Der Buchstabe kennzeichnet den Bausteinstatus/Netzwerk. Die x kennzeichnen die 
//Sprungmarkennummer in dezimaler Form.
//
//Ьber das Byte "byIntStatus" wird der Bausteinstatus (Statemachine) 
//gekennzeichnet:
//   0x10 SCHREIBE RESET (Synchron Reset)
//   0x20 START (neuen Sendeauftrag starten)
//   0x30 SENDEN (Sendeauftrag bearbeiten)
//   0x40 TLG QUITTUNG (Quittierung bearbeiten)
//   0x50 ABSCHLIEЯEN (Auftrag abschließen)
//   0x60 ERROR (Sendefehler und Warten auf Quittung)
//
//*******************************************************************************************
// Eingangsdaten konsistent lesen
//*******************************************************************************************
      L     #LADDR;
      T     #wLaddr;
//  DSTBLK zusammenbauen
      LAR1  P##anyDst;	// Any Pointer Anfangsadresse  
      L     W#16#1002;
      T     LW [AR1,P#0.0];	// Byte 0+1: Datentyp Byte  
      L     #IO_SIZE;
      T     LW [AR1,P#2.0];	// Byte 2+3: Länge 
      L     DINO;
      T     LW [AR1,P#4.0];	// Byte 4+5: DB-Nummer 
      TAR2;
      AD    DW#16#FFFFFF;
      L     P##arInputData;
      +D;
      T     LD [AR1,P#6.0];	// DWord 6: Speicherbereich + Offset im Speicherbereich
// Eingangsdaten lesen
      CALL  "DPRD_DAT" (
           LADDR                    := #wLaddr,
           RET_VAL                  := #iRetval,
           RECORD                   := #anyDst);
// RetVal auswerten
      L     #iRetval;
      L     0;
      ==I;
      JC    S001;
      L     #iRetval;
      T     #STATUS;	// schreibe STATUS = iRetVal DPRD_DAT
      JU    E100;
S001: NOP   0;
//*******************************************************************************************
// CONTROL aktualisieren
//*******************************************************************************************
      L     #CONTROL;
      T     #arOutputData[0];
//*******************************************************************************************
// Auftrag/Reset mit Fehler oder abgeschlossener Reset -> Handling Ausgänge
//*******************************************************************************************
      O     #REQ;
      O     #R;
      A     #ERROR;
      S     #xWait;
      A     #xFpReset;
      A     #DONE;
      S     #xWait;
      CLR;
      =     #DONE;
      =     #ERROR;
      L     0;
      T     #STATUS;
      AN    #REQ;
      AN    #R;
      R     #xWait;
      A     #xWait;
      JC    E100;
//*******************************************************************************************
// EN_R=0 während Datenempfang -> Synchron Reset anstoßen
//*******************************************************************************************
      A     #REQ;
      JC    I000;
      L     #bIntStatus;
      L     B#16#0;	// Datensendung aktiv?
      ==I;
      JC    I000;	// nein
      SET;
      =     #xResetBecauseAbort;	// ja -> REQ während Ьbertragung zurückgesetzt -> Synchron Reset anstoßen
I000: NOP   0;
//*******************************************************************************************
// Aufruf mit REQ=R=0 und keine fallende Flanke an REQ -> Baustein verlassen
//*******************************************************************************************
      O     #REQ;
      O     #R;
      O     #xResetBecauseAbort;
      JC    I010;
// Ausgangsparameter (Ausgangsdaten bleiben unverändert) und statische Variablen zurücksetzen
      CLR;
      =     #DONE;	// DONE 
      =     #ERROR;	// ERROR 
      =     #xFpRequest;
      =     #xFpReset;
      =     #xResetDone;
      =     #xResetBecauseAbort;
      L     0;
      T     #STATUS;	// STATUS
      T     #bIntStatus;
      T     #bAcknowledge;
      T     #bFrag;
      T     #bFragCounter;
      T     #iLenTrailer;
      JU    E100;	// Baustein verlassen
I010: NOP   0;
//*******************************************************************************************
// Eingangsparameter prüfen
//*******************************************************************************************
// Reset auch bei ungültigen Eingangsparametern möglich
      A     #R;
      ON    #REQ;
      JC    I024;
// DB_NO prüfen
      L     #DB_NO;
      L     0;
      <>I;	// Fehler bei DB_NO=0
      JC    I020;
      L     W#16#301;
      T     #STATUS;	// schreibe STATUS 0x0301
      JU    E100;	// Baustein verlassen
I020: NOP   0;
// LEN prüfen
      L     #LEN;
      L     0;
      ==I;	// Fehler bei LEN=0
      JC    I021;
      L     #LEN;
      L     1024;
      >I;	// Fehler bei LEN>1024
      JCN   I022;
I021: NOP   0;
      L     W#16#517;
      T     #STATUS;	// schreibe STATUS 0x0517
      JU    E100;	// Baustein verlassen
I022: NOP   0;
// IO_SIZE prüfen
      L     #IO_SIZE;
      L     0;
      ==I;	// Fehler bei IO_SIZE=0
      JC    I023;
      L     #IO_SIZE;
      L     60;
      >I;	// Fehler bei IO_SIZE>60
      JCN   I024;
I023: NOP   0;
      L     W#16#202;
      T     #STATUS;	// schreibe STATUS 0x0202
      JU    E100;	// Baustein verlassen
I024: NOP   0;
// keine Fehler an den Eingangsparametern -> STATUS zurücksetzen
      L     W#16#0;
      T     #STATUS;	// schreibe STATUS 0x0000
//*******************************************************************************************
// Aufruf mit R=1 (Reset immer möglich, unabhängig von REQ)
//*******************************************************************************************
      O     #R;	// R gesetzt?
      O     #xResetBecauseAbort;	// oder Reset durch fallende Flanke an REQ?
      JCN   I030;	// nein -> Flankenmerker R zurücksetzen 
      A     #xFpReset;	// Synchon Reset bereits gesartet?
      JC    I031;	// ja -> Reset bearbeiten
// neuen Reset anstoßen
      L     B#16#10;	// Int_Status = SCHREIBE RESET
      T     #bIntStatus;
      SET;
      =     #xFpReset;
      JU    I031;
I030: NOP   0;
      CLR;
      =     #xFpReset;	// Flankenmerker R zurücksetzen 
I031: NOP   0;
//*******************************************************************************************
// Aufruf mit REQ=1 (Senden nur mit R=0 möglich)
//*******************************************************************************************
      A     #xFpReset;	// Reset angestoßen?
      JC    I040;	// ja -> Synchron Reset bearbeiten
      AN    #REQ;	// REQ gesetzt?
      JC    E100;	// nein -> Baustein verlassen
      A     #DONE;	// Auftrag bereits bearbeitet
      JC    E100;	// Baustein verlassen
// neuen Auftrag anstoßen oder aktuellen Auftrag bearbeiten
      A     #xFpRequest;
      JC    I040;
      L     B#16#20;	// Int_Status = START
      T     #bIntStatus;
      SET;
      =     #xFpRequest;
I040: NOP   0;
//*******************************************************************************************
// Quittierungsbyte generieren
//*******************************************************************************************
      L     #arInputData[0];
      SRW   4;
      T     #bAcknowledge;	// Quittierungsbyte = Bit 4..7 von Eingangsbyte 0 
//*******************************************************************************************
// Bausteinstatus auswerten
//*******************************************************************************************
// Int_Status = SCHREIBE RESET
      L     B#16#10;
      L     #bIntStatus;
      ==I;
      JC    R000;
// Int_Status = START
      L     B#16#20;
      L     #bIntStatus;
      ==I;
      JC    S000;
// Int_Status = SENDEN
      L     B#16#30;
      L     #bIntStatus;
      ==I;
      JC    T000;
// Int_Status = TLQ QUITTUNG
      L     B#16#40;
      L     #bIntStatus;
      ==I;
      JC    Q000;
// Int_Status = ABSCHLIEЯEN
      L     B#16#50;
      L     #bIntStatus;
      ==I;
      JC    A000;
// Int_Status = ERROR
      L     B#16#60;
      L     #bIntStatus;
      ==I;
      JC    ER00;
// Int_Status nicht definiert = ENDE
      JU    E100;
NETWORK
TITLE = SCHREIBE RESET
R000: NOP   0;
//*******************************************************************************************
// "Reset abschließen" prüfen
//*******************************************************************************************
      A     #xResetDone;
      JC    R010;	// Quittung 0x08 prüfen
      JU    R020;	// Quittung 0x0C prüfen
R010: NOP   0;
//*******************************************************************************************
// Quittung 0x08 prüfen
//*******************************************************************************************
      L     #bAcknowledge;
      L     B#16#8;
      <>I;
      JC    R011;
      L     B#16#0;	// Int_Status = zurücksetzen
      T     #bIntStatus;
      CLR;
      =     #xResetDone;
      =     #xResetBecauseAbort;
R011: NOP   0;
      JU    E100;	// Baustein verlassen
R020: NOP   0;
//*******************************************************************************************
// Quittung 0x0C prüfen
//*******************************************************************************************
      L     #bAcknowledge;
      L     B#16#C;
      <>I;
      JC    R021;
// Ausgangsbyte 0 = CONTROL
      L     #CONTROL;
      L     B#16#F0;
      AW;
      L     B#16#8;	// Synchron Reset quittieren
      OW;
      T     #arOutputData[0];
      SET;
      =     #xResetDone;	// "Reset abschließen" setzen 
      =     #DONE;	// DONE setzen
      JU    R022;
R021: NOP   0;
// Ausgangsbyte 0 = CONTROL
      L     #CONTROL;
      L     B#16#F0;
      AW;
      L     B#16#B;	// Synchron Reset Quittierung anfordern
      OW;
      T     #arOutputData[0];
R022: NOP   0;
      JU    E100;	// Baustein verlassen
NETWORK
TITLE = START
// (network holds code this reader does not know; not shown)
//*******************************************************************************************
// Quittung 0x08 prüfen
//*******************************************************************************************
//*******************************************************************************************
// Fragmentanzahl berechnen und prüfen
//*******************************************************************************************
// Zwischenwert 1 = Dividend
// Zwischenwert 2 = Divisor
// Dividend / Divisor -> Quotient ohne Divisionsrest
// Dividend / Divisor -> Divisionsrest = Länge des Trailer
// Fragmentanzahl=1 ?
//*******************************************************************************************
// Schreibe Header/Trailer kombiniert
//*******************************************************************************************
// DONE zurücksetzen
// Ausgangsbyte 0 = CONTROL
// Int_Status = TLQ QUITTUNG setzen
//*******************************************************************************************
// Schreibe Header
//*******************************************************************************************
// DONE zurücksetzen
// Ausgangsbyte 0 = CONTROL
// Fragmentzähler auf 1 setzen
// Int_Status = SENDEN setzen
//*******************************************************************************************
// gemeinsame Sendedaten Header/Trailer kombiniert / Header generieren
//*******************************************************************************************
// Ausgangsbyte 1 = 0x00 
// Ausgangsbyte 2+3 = LEN 
// Ausgangsbyte 4-16 = SRCBLK zusammenbauen
// Ausgangsbyte 4-16 = DSTBLK zusammenbauen
// STATUS schreiben
NETWORK
TITLE = SENDEN
T000: NOP   0;
//*******************************************************************************************
// Quittung = letzte Fragmentnummer prüfen
//*******************************************************************************************
// Fragmentnummer steht in Bit0..2 der Quittierung
      L     #bAcknowledge;
      L     B#16#7;
      AW;
      T     #wTemp1;
// Fragmentnummer = Fragmentzähler & 0x07
      L     #bFragCounter;
      L     B#16#7;
      AW;
      T     #wTemp2;
// vergleiche Quittierung mit Fragmentnummer
      L     #wTemp1;
      L     #wTemp2;
      ==I;
      JC    T010;
      JU    E100;	// Baustein verlassen
T010: NOP   0;
// Fragmentzähler um 1 inkrementieren
      L     #bFragCounter;
      L     1;
      +I;
      T     #bFragCounter;
//*******************************************************************************************
// Fragmentzähler = Fragmentanzahl ?
//*******************************************************************************************
      L     #bFrag;
      L     #bFragCounter;
      ==I;
      JC    T020;	// schreibe Trailer
      JU    T030;	// schreibe Fragment
T020: NOP   0;
//*******************************************************************************************
// Schreibe Trailer
//*******************************************************************************************
// Ausgangsbyte 0 = CONTROL
      L     #CONTROL;
      L     B#16#F0;
      AW;
      L     B#16#A;	// Datensendung ьber RS232 vorbereiten -> Trailer
      OW;
      T     #arOutputData[0];
//  Sendedaten Trailer generieren
      L     #iLenTrailer;
      T     #wTemp1;	// Byte 2+3: Trailer Länge 
      T     #wTemp2;	// Byte 2+3: Trailer Länge 
// Int_Status = TLQ QUITTUNG setzen
      L     B#16#40;
      T     #bIntStatus;	// Int_Status = TLQ QUITTUNG
      JU    T050;	// gemeinsame Sendedaten Trailer/Fragment generieren
T030: NOP   0;
//*******************************************************************************************
// Schreibe Fragment
//*******************************************************************************************
// Ausgangsbyte 0 = Fragmentnummer = Fragmentzähler & 0x07
      L     #CONTROL;	// Datensendung ьber RS232 vorbereiten -> Fragment
      L     B#16#F0;
      AW;
      L     #bFragCounter;
      SLW   13;
      SRW   13;
      OW;
      L     B#16#F7;	// Ausmaskieren des Steuerbits
      AW;
      T     #arOutputData[0];
//  Sendedaten Fragment generieren
      L     #IO_SIZE;
      L     1;
      -I;
      T     #wTemp1;	// Byte 2+3: Fragmentlänge = IO_SIZE - 1 Byte
      T     #wTemp2;	// Byte 2+3: Fragmentlänge = IO_SIZE - 1 Byte
      JU    T050;	// gemeinsame Sendedaten Trailer/Fragment generieren
T050: NOP   0;
//*******************************************************************************************
// gemeinsame Sendedaten Trailer/Fragment generieren
//*******************************************************************************************
      L     #bFragCounter;
      L     2;
      -D;
      L     #IO_SIZE;
      DEC   1;
      *D;
      L     #IO_SIZE;
      +D;
      L     #DBB_NO;
      +D;
      L     4;
      -D;
      SLD   3;
      T     #dwTemp1;	// Byte 8+9: Offset im Sende-DB 
      L     8;
      T     #dwTemp2;	// Byte 8+9: Offset im Ausgangsdatenbereich ist 1 Byte = 8 Bit
      JU    E000;
NETWORK
TITLE = TLQ QUITTUNG
Q000: NOP   0;
//*******************************************************************************************
// Quittung 0x0A prüfen
//*******************************************************************************************
      L     #bAcknowledge;
      L     B#16#A;
      ==I;
      JC    Q010;
      JU    E100;	// Baustein verlassen
Q010: NOP   0;
// Ausgangsbyte 0 = CONTROL
      L     #CONTROL;
      L     B#16#F0;
      AW;
      L     B#16#8;	// Daten ьber RS232 senden
      OW;
      T     #arOutputData[0];
// Int_Status = ABSCHLIEЯEN setzen und Baustein verlassen        
      L     B#16#50;
      T     #bIntStatus;	// Int_Status = ABSCHLIEЯEN
      JU    E100;	// Baustein verlassen
NETWORK
TITLE = ERROR
ER00: NOP   0;
      L     #bAcknowledge;
      L     B#16#8;
      ==I;
      JC    ER10;
      JU    E100;
//*******************************************************************************************
// Quittung 0x08 prüfen
//*******************************************************************************************
ER10: NOP   0;
// STATUS schreiben
      L     #wStatusMem;
      T     #STATUS;	// schreibe zwischengespeicherten STATUS
// Int_Status zurücksetzen und Baustein verlassen
      L     B#16#0;
      T     #bIntStatus;	// Int_Status zurücksetzen
      L     #CONTROL;
      L     B#16#F0;
      AW;
      L     B#16#8;	// CP Ruhezustand quittieren
      OW;
      T     #arOutputData[0];
      JU    E100;	// Baustein verlassen
NETWORK
TITLE = ABSCHLIEЯEN
A000: NOP   0;
      L     #bAcknowledge;
      L     B#16#8;
      ==I;
      JC    A010;
      L     #bAcknowledge;
      L     B#16#D;
      ==I;
      JC    A020;
      L     #bAcknowledge;
      L     B#16#E;
      ==I;
      JC    A030;
      JU    E100;	// Baustein verlassen
//*******************************************************************************************
// Quittung 0x08 prüfen
//*******************************************************************************************
A010: NOP   0;
// STATUS schreiben
      L     W#16#0;
      T     #STATUS;	// schreibe STATUS 0x0000
// DONE setzen
      SET;
      =     #DONE;
// Int_Status zurücksetzen und Baustein verlassen
      L     B#16#0;
      T     #bIntStatus;	// Int_Status zurücksetzen
      JU    E100;	// Baustein verlassen
//****************************************************************************************
// Quittung 0x0D prüfen
//*******************************************************************************************
A020: NOP   0;
// Ausgangsbyte 0 = CONTROL
      L     #CONTROL;
      L     B#16#F0;
      AW;
      L     B#16#D;	// signalisiere ungültige Länge
      OW;
      T     #arOutputData[0];
// Fehlerstatus zwischenspeichern
      L     W#16#517;
      T     #wStatusMem;
// Int_Status = ERROR setzen und Baustein verlassen        
      L     B#16#60;
      T     #bIntStatus;	// Int_Status = ERROR
      JU    E100;	// Baustein verlassen
//****************************************************************************************
// Quittung 0x0E prüfen
//*******************************************************************************************
A030: NOP   0;
// Ausgangsbyte 0 = CONTROL
      L     #CONTROL;
      L     B#16#F0;
      AW;
      L     B#16#E;	// signalisiere Ьbertragung fehlgeschlagen
      OW;
      T     #arOutputData[0];
// Fehlerstatus zwischenspeichern
      L     W#16#70A;
      T     #wStatusMem;
// Int_Status = ERROR setzen und Baustein verlassen        
      L     B#16#60;
      T     #bIntStatus;	// Int_Status = ERROR
      JU    E100;	// Baustein verlassen
NETWORK
TITLE = ENDE
E000: NOP   0;
//*******************************************************************************************
// Daten kopieren
//*******************************************************************************************
//  SRCBLK zusammenbauen
      LAR1  P##anyScr;	// Any Pointer Anfangsadresse  
      L     W#16#1002;
      T     LW [AR1,P#0.0];	// Byte 0+1: Datentyp Byte 
      L     #wTemp1;
      T     LW [AR1,P#2.0];	// Byte 2+3: Länge 
      L     #DB_NO;
      T     LW [AR1,P#4.0];	// Byte 4+5: Sende-DB Nummer 
      L     #dwTemp1;
      T     LD [AR1,P#6.0];	// Byte 7+8+9: Offset im Sende-DB 
      L     B#16#84;
      T     LB [AR1,P#6.0];	// Byte 6: Speicherbereich DB
//  DSTBLK zusammenbauen
      LAR1  P##anyDst;	// Any Pointer Anfangsadresse  
      L     W#16#1002;
      T     LW [AR1,P#0.0];	// Byte 0+1: Datentyp Byte  
      L     #wTemp2;
      T     LW [AR1,P#2.0];	// Byte 2+3: Länge 
      L     DINO;
      T     LW [AR1,P#4.0];	// Byte 4+5: DB-Nummer 
      TAR2;
      AD    DW#16#FFFFFF;
      L     P##arOutputData;
      +D;
      L     #dwTemp2;
      +D;
      T     LD [AR1,P#6.0];	// DWord 6: Speicherbereich + Offset im Speicherbereich
// Sendedaten auf Ausgangsdaten umkopieren (nicht verwendete Ausgangsdaten behalten alten Wert)
      CALL  "BLKMOV" (
           SRCBLK                   := #anyScr,
           RET_VAL                  := #iRetval,
           DSTBLK                   := #anyDst);
// RetVal auswerten
      L     #iRetval;
      L     0;
      ==I;
      JC    E001;
      L     #iRetval;
      T     #STATUS;	// schreibe STATUS = iRetVal BLKMOV
E001: NOP   0;
E100: NOP   0;
//*******************************************************************************************
// Ausgangsdaten konsistent schreiben
//*******************************************************************************************
      L     #LADDR;
      T     #wLaddr;
//  DSTBLK zusammenbauen
      LAR1  P##anyScr;	// Any Pointer Anfangsadresse  
      L     W#16#1002;
      T     LW [AR1,P#0.0];	// Byte 0+1: Datentyp Byte  
      L     #IO_SIZE;
      T     LW [AR1,P#2.0];	// Byte 2+3: Länge 
      L     DINO;
      T     LW [AR1,P#4.0];	// Byte 4+5: DB-Nummer 
      TAR2;
      AD    DW#16#FFFFFF;
      L     P##arOutputData;
      +D;
      T     LD [AR1,P#6.0];	// DWord 6: Speicherbereich + Offset im Speicherbereich
// Ausgangsdaten schreiben
      CALL  "DPWR_DAT" (
           LADDR                    := #wLaddr,
           RECORD                   := #anyScr,
           RET_VAL                  := #iRetval);
// RetVal auswerten
      L     #iRetval;
      L     0;
      ==I;
      JC    S002;
      L     #iRetval;
      T     #STATUS;	// schreibe STATUS = iRetVal DPWR_DAT
S002: NOP   0;
//*******************************************************************************************
// schreibe CONTROL
//*******************************************************************************************
// schreibe CONTROL
      L     #arOutputData[0];	// CONTROL (Bit 0..3) 
      T     #CONTROL;
//*******************************************************************************************
// ERROR Bit steuern und auf BIE (Statuswort, Bit 8) abbilden
//*******************************************************************************************
// ERROR steuern
      L     #STATUS;
      L     B#16#0;	// STATUS = 0x0000 -> kein Fehler
      ==I;
      JC    E110;
      L     #STATUS;
      L     W#16#8181;	// STATUS = 0x8181 -> Senden
      ==I;
      JC    E110;
      SET;
      =     #ERROR;	// STATUS = Fehler -> ERROR setzen
      JU    E111;
E110: NOP   0;
      CLR;
      =     #ERROR;	// STATUS = kein Fehler -> ERROR zurücksetzen
E111: NOP   0;
// BIE steuern
      AN    #ERROR;
      SAVE;	// BIE=VKE
END_FUNCTION_BLOCK

FUNCTION_BLOCK "RECEIVE"	// FB 61
TITLE = RECEIVE
//Histoy:
//V1.0   erste Version
//V1.2   Ьbergabe BLKMOV RetVal an Status
//       Reset auch bei fehlerhaften Eingangsparametern möglich
//       Ausgangsbits stehen nur für einen SPS-Zyklus an
//V1.3   Korrektur Verarbeitung des empfangenen DataOffset
//V2.0   Prozessdatenzugriff auf SFC14 und PAB umgestellt
//V2.1   Korrektur im SEND-Baustein, keine Дnderung RECEIVE-Baustein
VERSION : 2.1
VAR_INPUT
  EN_R : BOOL ;	//Freigabe für Daten lesen
  R : BOOL ;	//Synchron Reset auslösen
  LADDR : INT ;	//logische Basisadresse des CP - entspricht der Adresse aus der HW-Konfiguration
  DB_NO : INT ;	//Datenbausteinnummer - Nummer des Empfangs-DB (>0)
  DBB_NO : INT ;	//Datenbytenummer - Empfangsdaten ab Datenbyte
  IO_SIZE : WORD ;	//parametrierte IO Größe des Moduls
END_VAR
VAR_OUTPUT
  LEN : INT ;	//Länge des empfangenen Telegramms in Byte (>0 und <1025)
  NDR : BOOL ;	//Auftrag fertig ohne Fehler, Daten empfangen, Parameter STATUS=00h
  ERROR : BOOL ;	//Auftrag fertig mit Fehler, Parameter STATUS enthält die Fehlerinformation
  STATUS : WORD ;	//Spezifikation des Fehlers bei ERROR=1
END_VAR
VAR_IN_OUT
  CONTROL : BYTE ;	//geteilter Speicher: Sendebaustein Bit 0..3, Empfangsbaustein Bit 4-7
END_VAR
VAR
  bIntStatus : BYTE ;	//interner Bausteinstatus
  xFpReset : BOOL ;	//Hilfsbit zur Erkennung einer steigenden Flanke an R
  xResetDone : BOOL ;	//Fertigmeldung Synchron Reset (Statemachine Bit)
  bFragNr : BYTE ;	//Fragmentnummer
  iLen : INT ;	//gelieferte Länge im Header bzw. Header/Trailer kombiniert
  iLenRead : INT ;	//Anzahl der bisher gelesenen Bytes
  iTeleOffset : INT ;	//geliefertes Telegramm Offset im Header bzw. Header/Trailer kombiniert
  wReturnValue : WORD ;	//geliefertes Return Value im Header bzw. Header/Trailer kombiniert
  xResetBecauseAbort : BOOL ;	//Reset durch fallende Flanke an EN_R ausgelöst
  iFragCounter : INT ;	//Fragmentzähler
  xWait : BOOL ;	//warte nach fertigem Reset oder Auftrag mit Fehler auf FALS an EN_R und R
  arInputData : ARRAY  [0 .. 59 ] OF BYTE ;
  arOutputData : ARRAY  [0 .. 0 ] OF BYTE ;
END_VAR
VAR_TEMP
  wTemp1 : WORD ;
  wTemp2 : WORD ;
  dwTemp1 : DWORD ;
  dwTemp2 : DWORD ;
  anyScr : ANY ;
  anyDst : ANY ;
  iRetval : INT ;
  wLaddr : WORD ;
END_VAR
BEGIN
NETWORK
TITLE = INIT
//
//Sprungmarken Definition:
//   Ixxx INIT
//   Rxxx SCHREIBE RESET
//   E8xx Eingangsbyte=Fragmentnummer=0x08
//   EAxx Eingangsbyte=Fragmentnummer=0x0A
//   E9xx Eingangsbyte=Fragmentnummer=0x09
//   Hxxx HEADER EMPFANGEN
//   Exxx ENDE
//Der Buchstabe kennzeichnet den Bausteinstatus/Netzwerk. Die x kennzeichnen die 
//Sprungmarkennummer in dezimaler Form.
//
//Ьber das Byte "byIntStatus" wird der Bausteinstatus (Statemachine) 
//gekennzeichnet:
//   0x00 LEERLAUF (lese Header/Trailer oder Header oder warte auf Daten)
//   0x10 SCHREIBE RESET (Synchron Reset)
//   0x20 HEADER EMPFANGEN (lese Fragment oder Trailer)
//   0x30 AUFTRAG ABSCHLIEЯEN
// 
//*******************************************************************************************
// Eingangsdaten konsistent lesen
//*******************************************************************************************
      L     #LADDR;
      T     #wLaddr;
//  DSTBLK zusammenbauen
      LAR1  P##anyDst;	// Any Pointer Anfangsadresse  
      L     W#16#1002;
      T     LW [AR1,P#0.0];	// Byte 0+1: Datentyp Byte  
      L     #IO_SIZE;
      T     LW [AR1,P#2.0];	// Byte 2+3: Länge 
      L     DINO;
      T     LW [AR1,P#4.0];	// Byte 4+5: DB-Nummer 
      TAR2;
      AD    DW#16#FFFFFF;
      L     P##arInputData;
      +D;
      T     LD [AR1,P#6.0];	// DWord 6: Speicherbereich + Offset im Speicherbereich
// Eingangsdaten lesen
      CALL  "DPRD_DAT" (
           LADDR                    := #wLaddr,
           RET_VAL                  := #iRetval,
           RECORD                   := #anyDst);
// RetVal auswerten
      L     #iRetval;
      L     0;
      ==I;
      JC    S001;
      L     #iRetval;
      T     #STATUS;	// schreibe STATUS = iRetVal DPRD_DAT
      JU    E100;
S001: NOP   0;
//*******************************************************************************************
// CONTROL aktualisieren
//*******************************************************************************************
      L     #CONTROL;
      T     #arOutputData[0];
//*******************************************************************************************
// Auftrag/Reset mit Fehler oder abgeschlossener Reset -> Handling Ausgänge
//*******************************************************************************************
      O     #EN_R;
      O     #R;
      A     #ERROR;
      JCN   FE00;
      L     0;
      T     #STATUS;
      SET;
      =     #xWait;
FE00: NOP   0;
      A     #xFpReset;	// wenn Reset angestoßen
      A     #NDR;	// und bearbeitet
      S     #xWait;
      R     #NDR;
      AN    #EN_R;
      AN    #R;
      R     #xWait;
      A     #xWait;
      JC    E100;
//*******************************************************************************************
// EN_R=0 während Datenempfang -> Synchron Reset anstoßen
//*******************************************************************************************
      O     #EN_R;
      O     #NDR;
      JC    I000;
      L     #bIntStatus;
      L     B#16#0;	// Int_Status = LEERLAUF?
      ==I;
      JC    I000;
      SET;
      =     #xResetBecauseAbort;	// fallende Flanke an EN_R erkannt
I000: NOP   0;
//*******************************************************************************************
// Aufruf mit EN_R=R=0 und keine fallende Flanke an EN_R -> Baustein verlassen
//*******************************************************************************************
      O     #EN_R;
      O     #R;
      O     #xResetBecauseAbort;
      JC    I010;
// Ausgangsparameter (Ausgangsdaten bleiben unverändert) und statische Variablen zurücksetzen
      CLR;
      =     #NDR;	// NDR 
      =     #ERROR;	// ERROR 
      =     #xFpReset;
      =     #xResetDone;
      =     #xResetBecauseAbort;
      L     0;
      T     #LEN;	// LEN
      T     #STATUS;	// STATUS
      T     #bIntStatus;
      T     #bFragNr;
      T     #iLen;
      T     #iLenRead;
      T     #iTeleOffset;
      T     #wReturnValue;
      T     #iFragCounter;
//wenn kein Auftrag ansteht -> Idle Zustand an CP melden
      L     #CONTROL;
      L     B#16#F;
      AW;
      L     B#16#80;
      OW;
      T     #arOutputData[0];
      JU    E200;	// Baustein verlassen
I010: NOP   0;
//*******************************************************************************************
// Eingangsparameter prüfen
//*******************************************************************************************
// Reset auch bei ungültigen Eingangsparametern möglich
      A     #R;
      JC    I022;
// DB_NO prüfen
      L     #DB_NO;
      L     0;
      <>I;	// Fehler bei DB_NO=0
      JC    I020;
      L     W#16#301;
      T     #STATUS;	// schreibe STATUS 0x0301
      SET;
      =     #ERROR;	// ERROR setzen
      JU    E200;	// Baustein verlassen
I020: NOP   0;
// IO_SIZE prüfen
      L     #IO_SIZE;
      L     0;
      ==I;	// Fehler bei IO_SIZE=0
      JC    I021;
      L     #IO_SIZE;
      L     60;
      >I;	// Fehler bei IO_SIZE>60
      JCN   I022;
I021: NOP   0;
      L     W#16#202;
      T     #STATUS;	// schreibe STATUS 0x0202
      SET;
      =     #ERROR;	// ERROR setzen
      JU    E200;	// Baustein verlassen
I022: NOP   0;
// keine Fehler an den Eingangsparametern -> ERROR und STATUS zurücksetzen
      L     W#16#0;
      T     #STATUS;	// schreibe STATUS 0x0000
      CLR;
      =     #ERROR;	// ERROR zurücksetzen
//*******************************************************************************************
// Aufruf mit R=1 (Reset immer möglich, unabhängig von EN_R)
//*******************************************************************************************
      O     #R;	// R gesetzt?
      O     #xResetBecauseAbort;	// oder Reset durch fallende Flanke an EN_R?
      JCN   I030;	// nein -> Flankenmerker R zurücksetzen 
      A     #xFpReset;	// Synchon Reset bereits gesartet?
      JC    I031;	// ja -> Reset bearbeiten
// neuen Reset anstoßen
      L     B#16#10;	// Int_Status = SCHREIBE RESET
      T     #bIntStatus;
      SET;
      =     #xFpReset;
      JU    I031;
I030: NOP   0;
      CLR;
      =     #xFpReset;	// Flankenmerker R zurücksetzen 
I031: NOP   0;
      A     #xFpReset;	// wenn Reset angestoßen
      A     #NDR;	// und bearbeitet
      JC    E100;	// --> Bausteinende
//*******************************************************************************************
// Aufruf mit EN_R=1 (Empfang nur mit R=0 möglich)
//*******************************************************************************************
      A     #xFpReset;	// Reset angestoßen?
      JC    I040;	// ja -> Synchron Reset bearbeiten
      AN    #EN_R;	// EN_R gesetzt?
      JC    E200;	// nein -> Baustein verlassen
      A     #NDR;	// Auftrag abgeschlossen?
      JCN   I040;	// nein -> Auftrag bearbeiten
// Auftrag bearbeitet -> Ausgangsparameter zurücksetzen
      L     0;
      T     #LEN;	// LEN
      T     #STATUS;	// STATUS
      T     #iLen;
      T     #iLenRead;
      T     #bIntStatus;	// Int_Status = LEERLAUF
      T     #iTeleOffset;
      T     #iFragCounter;
      CLR;
      =     #NDR;
I040: NOP   0;
//*******************************************************************************************
// Fragmentnummer bestimmen
//*******************************************************************************************
// logische Basisadresse in das Adressregister schreiben
      L     #arInputData[0];
      SLW   12;
      SRW   12;
      T     #bFragNr;	// Fragmentnummer = Bit 0..3 von Eingangsbyte 0 
//*******************************************************************************************
// Bausteinstatus / Eingangsbyte=Fragmentnummer auswerten
//*******************************************************************************************
// Int_Status = SCHREIBE RESET
      L     B#16#10;
      L     #bIntStatus;
      ==I;
      JC    R000;
// Int_Status = Eingangsbyte=Fragmentnummer=0x08
      L     #bFragNr;
      L     B#16#8;
      ==I;
      JC    E800;
// Int_Status = Eingangsbyte=Fragmentnummer=0x0A
      L     #bFragNr;
      L     B#16#A;
      ==I;
      JC    EA00;
// Int_Status = Eingangsbyte=Fragmentnummer=0x09
      L     #bFragNr;
      L     B#16#9;
      ==I;
      JC    E900;
// Int_Status = HEADER EMPFANGEN
      L     B#16#20;
      L     #bIntStatus;
      ==I;
      JC    H000;
// Int_Status nicht definiert
      L     W#16#407;
      T     #STATUS;	// schreibe STATUS 0x0407
      JU    E200;	// Baustein verlassen
NETWORK
TITLE = SCHREIBE RESET
R000: NOP   0;
//*******************************************************************************************
// "Reset abschließen" prüfen
//*******************************************************************************************
      A     #xResetDone;
      JC    R010;	// Fragmentnummer 0x08 prüfen
      JU    R020;	// Fragmentnummer 0x0C prüfen
R010: NOP   0;
//*******************************************************************************************
// Fragmentnummer 0x08 prüfen
//*******************************************************************************************
      L     #bFragNr;
      L     B#16#8;
      <>I;
      JC    R011;
      L     B#16#0;	// Int_Status = Leerlauf
      T     #bIntStatus;
      CLR;
      =     #xResetDone;
      =     #xResetBecauseAbort;
      SET;
      =     #NDR;
R011: NOP   0;
      JU    E200;	// Baustein verlassen
R020: NOP   0;
//*******************************************************************************************
// Fragmentnummer 0x0C prüfen
//*******************************************************************************************
      L     #bFragNr;
      L     B#16#C;
      <>I;
      JC    R021;
// Ausgangsbyte 0 = CONTROL
      L     #CONTROL;
      L     B#16#F;
      AW;
      L     B#16#80;	// Synchron Reset quittieren
      OW;
      T     #arOutputData[0];
      SET;
      =     #xResetDone;	// "Reset abschließen" setzen 
      JU    R022;
R021: NOP   0;
// Ausgangsbyte 0 = CONTROL
      L     #CONTROL;
      L     B#16#F;
      AW;
      L     B#16#B0;	// Synchron Reset Quittierung anfordern
      OW;
      T     #arOutputData[0];
R022: NOP   0;
      JU    E200;	// Baustein verlassen
NETWORK
TITLE = Eingangsbyte=Fragmentnummer=0x08
E800: NOP   0;
//*******************************************************************************************
// Prüfung ob Leerlauf oder Auftrag abschließen
//*******************************************************************************************
      L     B#16#30;	// Int_Status = AUFTRAG ABSCHLIEЯEN?
      L     #bIntStatus;
      ==I;
      JC    E810;	// ja -> Auftrag abschließen
      JU    E100;	// nein -> Ausgangsbyte 0 schreiben
E810: NOP   0;
//*******************************************************************************************
// Auftrag abschließen
//*******************************************************************************************
// Ausgangsparameter für einen SPS-Zyklus setzen
      L     #iLen;
      T     #LEN;	// LEN = Länge aus Header Daten
      L     #wReturnValue;
      T     #STATUS;	// STATUS = Return Value aus Header Daten
      SET;
      =     #NDR;
      JU    E100;	// Ausgangsbyte 0 schreiben
NETWORK
TITLE = Eingangsbyte=Fragmentnummer=0x0A
EA00: NOP   0;
//*******************************************************************************************
// Prüfung ob Trailer oder Header/Trailer kombiniert oder bereits bearbeitet
//*******************************************************************************************
      L     B#16#30;	// Int_Status = AUFTRAG ABSCHLIEЯEN?
      L     #bIntStatus;
      ==I;
      JC    E200;	// ja -> Baustein verlassen
      L     B#16#20;	// Int_Status = HEADER EMPFANGEN?
      L     #bIntStatus;
      ==I;
      JC    EA10;	// lese Trailer
      JU    EA20;	// lese Header/Trailer kombiniert
EA10: NOP   0;
//*******************************************************************************************
// lese Trailer
//*******************************************************************************************
// SRCBLK / DSTBLK zusammenbauen
      L     8;	// 1 Byte Header
      T     #dwTemp1;	// Byte 8+9: Offset im Eingangsdatenbereich
      L     #iLen;
      L     #iLenRead;
      -I;
      T     #wTemp1;	// Byte 2+3: Länge im Eingangsdatenbereich
      T     #wTemp2;	// Byte 2+3: Länge im Empfangs-DB
      L     #DBB_NO;
      L     #iLenRead;
      +D;
      SLD   3;
      T     #dwTemp2;	// Byte 8+9: Offset im Empfangs-DB
      JU    EA50;	// Auftragsabschluss anstoßen
EA20: NOP   0;
//*******************************************************************************************
// lese Header/Trailer kombiniert
//*******************************************************************************************
// Eingangsbyte 2+3 = Anzahl Datenbytes + 2
      L     #arInputData[2];
      SLW   8;
      L     #arInputData[3];
      OW;
      L     2;
      -I;
      T     #iLen;
// Eingangsbyte 1 = prüfe ob Telegramm mit oder ohne Offset
      L     #arInputData[1];
      L     B#16#4;	// Offset vorhanden?
      ==I;
      JC    EA21;	// ja
      L     #arInputData[1];
      L     B#16#0;	// Offset<>0?
      <>I;
      JC    E200;	// ja -> ungültiger Offset -> Baustein verlassen
// Eingangsbyte 4+5 = Return Value
      L     #arInputData[4];
      SLW   8;
      L     #arInputData[5];
      OW;
      T     #wReturnValue;
      JU    EA22;
EA21: NOP   0;
// Eingangsbyte 4+5 = Telegramm Offset
      L     2;	// Nutzdaten sind um 2 Byte nach hinten verschoben bei Offset<>0
      T     #iTeleOffset;
// Eingangsbyte 6+7 = Return Value
      L     #arInputData[6];
      SLW   8;
      L     #arInputData[7];
      OW;
      T     #wReturnValue;
EA22: NOP   0;
// SRCBLK / DSTBLK zusammenbauen
      L     6;	// 6 Byte Header
      L     #iTeleOffset;	// + mögliches Offset definiert durch Eingangsdaten
      +D;
      SLD   3;
      T     #dwTemp1;	// Byte 8+9: Offset im Eingangsdatenbereich
      L     #iLen;
      T     #wTemp1;	// Byte 2+3: Länge im Eingangsdatenbereich
      T     #wTemp2;	// Byte 2+3: Länge im Empfangs-DB
      L     #arInputData[4];	// Telegrammoffset 
      SLW   8;
      L     #arInputData[5];
      OW;
      L     #DBB_NO;
      +I;
      L     #iLenRead;
      +D;
      SLD   3;
      T     #dwTemp2;	// Byte 7+8+9: Offset im Empfangs-DB
      JU    EA50;	// Auftragsabschluss anstoßen
EA50: NOP   0;
//*******************************************************************************************
// Auftragsabschluss anstoßen
//*******************************************************************************************
      L     B#16#30;	// Int_Status = AUFTRAG ABSCHLIEЯEN
      T     #bIntStatus;
      JU    E000;	// Daten kopieren
NETWORK
TITLE = Eingangsbyte=Fragmentnummer=0x09
E900: NOP   0;
//*******************************************************************************************
// Prüfung ob Header bereits gelesen wurde
//*******************************************************************************************
      L     B#16#20;	// Int_Status = HEADER EMPFANGEN?
      L     #bIntStatus;
      ==I;
      JC    E200;	// ja -> Baustein verlassen
//*******************************************************************************************
// lese Header
//*******************************************************************************************
// Eingangsbyte 2+3 = Anzahl Datenbytes + 2
      L     #arInputData[2];
      SLW   8;
      L     #arInputData[3];
      OW;
      L     2;
      -I;
      T     #iLen;
// Eingangsbyte 1 = prüfe ob Telegramm mit oder ohne Offset
      L     #arInputData[1];
      L     B#16#4;	// Offset vorhanden?
      ==I;
      JC    E921;	// ja
      L     #arInputData[1];
      L     B#16#0;	// Offset<>0?
      <>I;
      JC    E900;	// ja -> ungültiger Offset -> Baustein verlassen
// Eingangsbyte 4+5 = Return Value
      L     #arInputData[4];
      SLW   8;
      L     #arInputData[5];
      OW;
      T     #wReturnValue;
      JU    E922;
E921: NOP   0;
// Eingangsbyte 4+5 = Telegramm Offset
      L     2;	// Nutzdaten sind um 2 Byte nach hinten verschoben bei Offset<>0
      T     #iTeleOffset;
// Eingangsbyte 6+7 = Return Value
      L     #arInputData[6];
      SLW   8;
      L     #arInputData[7];
      OW;
      T     #wReturnValue;
E922: NOP   0;
// SRCBLK / DSTBLK zusammenbauen
      L     6;	// 6 Byte Header
      L     #iTeleOffset;	// + mögliches Offset definiert durch Eingangsdaten
      +D;
      T     #wTemp1;	// = Offset
      SLD   3;
      T     #dwTemp1;	// Byte 8+9: Offset im Eingangsdatenbereich
      L     #IO_SIZE;
      L     #wTemp1;
      -I;
      T     #wTemp1;	// Byte 2+3: Länge im Eingangsdatenbereich
      T     #wTemp2;	// Byte 2+3: Länge im Empfangs-DB
      L     #arInputData[4];	// Telegrammoffset 
      SLW   8;
      L     #arInputData[5];
      OW;
      L     #DBB_NO;
      +I;
      L     #iLenRead;
      +D;
      SLD   3;
      T     #dwTemp2;	// Byte 7+8+9: Offset im Empfangs-DB
//*******************************************************************************************
// Auftragsabschluss anstoßen
//*******************************************************************************************
      L     B#16#20;	// Int_Status = HEADER EMPFANGEN
      T     #bIntStatus;
      JU    E000;	// Daten kopieren
NETWORK
TITLE = HEADER EMPFANGEN
H000: NOP   0;
//*******************************************************************************************
// Prüfung ob Fragment bereits gelesen wurde
//*******************************************************************************************
      L     #bFragNr;
      L     #iFragCounter;
      ==I;
      JC    E100;	// Ausgangsbyte 0 schreiben
      L     #bFragNr;
      T     #iFragCounter;
//*******************************************************************************************
// lese Fragment
//*******************************************************************************************
// SRCBLK / DSTBLK zusammenbauen
      L     8;	// 1 Byte Header
      T     #dwTemp1;	// Byte 8+9: Offset im Eingangsdatenbereich
      L     #IO_SIZE;	// Fragment hat immer die Größe IO_SIZE-1
      L     1;
      -I;
      T     #wTemp1;	// Byte 2+3: Länge im Eingangsdatenbereich
      T     #wTemp2;	// Byte 2+3: Länge im Empfangs-DB
      L     #DBB_NO;
      L     #iLenRead;
      +D;
      SLD   3;
      T     #dwTemp2;	// Byte 8+9: Offset im Empfangs-DB
      JU    E000;	// Daten kopieren
NETWORK
TITLE = ENDE
E000: NOP   0;
//*******************************************************************************************
// Daten kopieren
//*******************************************************************************************
//  SRCBLK zusammenbauen
      LAR1  P##anyScr;	// Any Pointer Anfangsadresse  
      L     W#16#1002;
      T     LW [AR1,P#0.0];	// Byte 0+1: Datentyp Byte 
      L     #wTemp1;
      T     LW [AR1,P#2.0];	// Byte 2+3: Länge 
      L     DINO;
      T     LW [AR1,P#4.0];	// Byte 4+5: DB-Nummer 
      TAR2;
      AD    DW#16#FFFFFF;
      L     P##arInputData;
      +D;
      L     #dwTemp1;
      +D;
      T     LD [AR1,P#6.0];	// DWord 6: Speicherbereich + Offset im Speicherbereich
//  DSTBLK zusammenbauen
      LAR1  P##anyDst;	// Any Pointer Anfangsadresse  
      L     W#16#1002;
      T     LW [AR1,P#0.0];	// Byte 0+1: Datentyp Byte  
      L     #wTemp2;
      T     LW [AR1,P#2.0];	// Byte 2+3: Länge 
      L     #DB_NO;
      T     LW [AR1,P#4.0];	// Byte 4+5: Empfangs-DB 
      L     #dwTemp2;
      T     LD [AR1,P#6.0];	// Byte 7+8+9: Offset im Empfangs-DB
      L     B#16#84;
      T     LB [AR1,P#6.0];	// Byte 6: Speicherbereich DB
// Eingangsdaten in Empfangs-DB umkopieren
      CALL  "BLKMOV" (
           SRCBLK                   := #anyScr,
           RET_VAL                  := #iRetval,
           DSTBLK                   := #anyDst);
// RetVal auswerten
      L     #iRetval;
      L     0;
      ==I;
      JC    E001;
      L     #iRetval;
      T     #STATUS;	// schreibe STATUS = iRetVal BLKMOV
E001: NOP   0;
// Anzahl der bereits kopierten/empfangenen Datenbytes aktualisieren
      L     #iLenRead;
      L     #wTemp2;	// Anzahl der in den DB geschriebenen Datenbytes
      +I;
      T     #iLenRead;
E100: NOP   0;
//*******************************************************************************************
// schreibe Ausgangsbyte 0
//*******************************************************************************************
//verknüpfe Controlbyte mit Fragmentnummer  
      L     #CONTROL;
      L     B#16#F;
      AW;
      L     #bFragNr;
      SLW   4;
      OW;
      T     #arOutputData[0];	// Ausgangsbyte 0 (Bit 4..7) 
E200: NOP   0;
//*******************************************************************************************
// schreibe CONTROL
//*******************************************************************************************
      L     #LADDR;
      SLD   3;
      LAR1;
// schreibe CONTROL
      L     #arOutputData[0];	// CONTROL (Bit 4..7) 
      T     #CONTROL;
      T     PQB [AR1,P#0.0];
//*******************************************************************************************
// ERROR Bit steuern und auf BIE (Statuswort, Bit 8) abbilden
//*******************************************************************************************
// ERROR steuern
      L     #STATUS;
      L     B#16#0;	// STATUS = 0x0000 -> kein Fehler
      ==I;
      JC    E110;
      SET;
      =     #ERROR;	// STATUS = Fehler -> ERROR setzen
      JU    E111;
E110: NOP   0;
      CLR;
      =     #ERROR;	// STATUS = kein Fehler -> ERROR zurücksetzen
E111: NOP   0;
// BIE steuern
      AN    #ERROR;
      SAVE;	// BIE=VKE
END_FUNCTION_BLOCK

// FB 72: know-how protected block, not included

FUNCTION "RS485_1" : VOID	// FC 1
VERSION : 0.1
VAR_TEMP
  S_PRIVOD_1R : REAL ;
  S_PRIVOD_2R : REAL ;
END_VAR
BEGIN
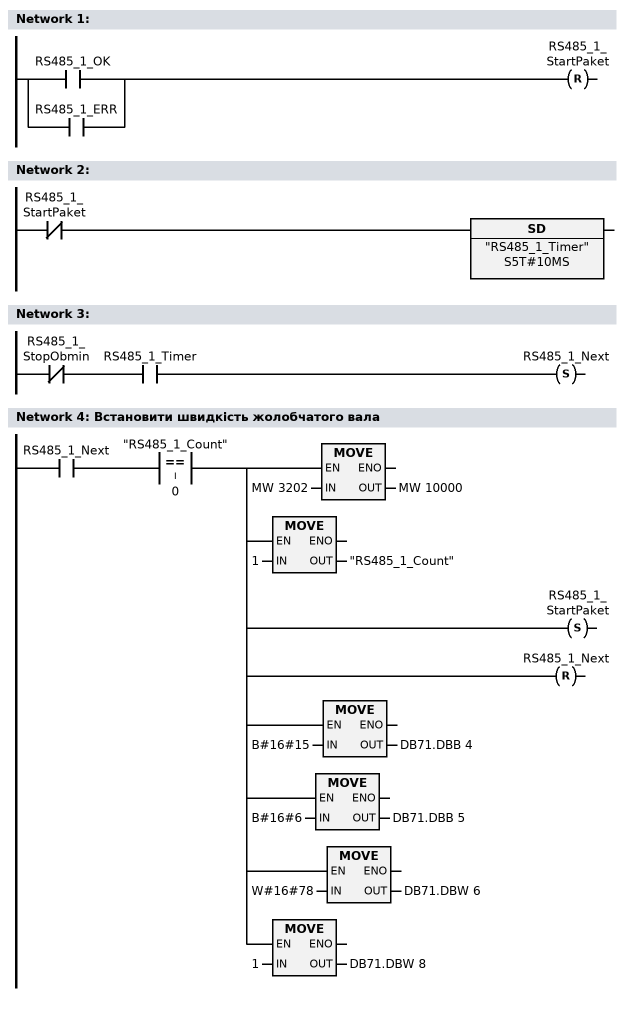
NETWORK
TITLE =
      O     "RS485_1_OK";
      O     "RS485_1_ERR";
      R     "RS485_1_StartPaket";
NETWORK
TITLE =
      AN    "RS485_1_StartPaket";
      L     S5T#10MS;
      SD    "RS485_1_Timer";
NETWORK
TITLE =
      AN    "RS485_1_StopObmin";
      A     "RS485_1_Timer";
      S     "RS485_1_Next";
NETWORK
TITLE = Встановити швидкість жолобчатого вала
      A     "RS485_1_Next";
      A(;
      L     "RS485_1_Count";
      L     0;
      ==I;
      );
      =     L 8.0;
      A     L 8.0;
      JNB   _001;
      L     MW 3202;
      T     MW 10000;
_001: NOP   0;
      A     L 8.0;
      JNB   _002;
      L     1;
      T     "RS485_1_Count";
_002: NOP   0;
      A     L 8.0;
      BLD   102;
      S     "RS485_1_StartPaket";
      A     L 8.0;
      BLD   102;
      R     "RS485_1_Next";
      A     L 8.0;
      JNB   _003;
      L     B#16#15;
      T     DB71.DBB 4;
_003: NOP   0;
      A     L 8.0;
      JNB   _004;
      L     B#16#6;
      T     DB71.DBB 5;
_004: NOP   0;
      A     L 8.0;
      JNB   _005;
      L     W#16#78;
      T     DB71.DBW 6;
_005: NOP   0;
      A     L 8.0;
      JNB   _006;
      L     1;
      T     DB71.DBW 8;
_006: NOP   0;
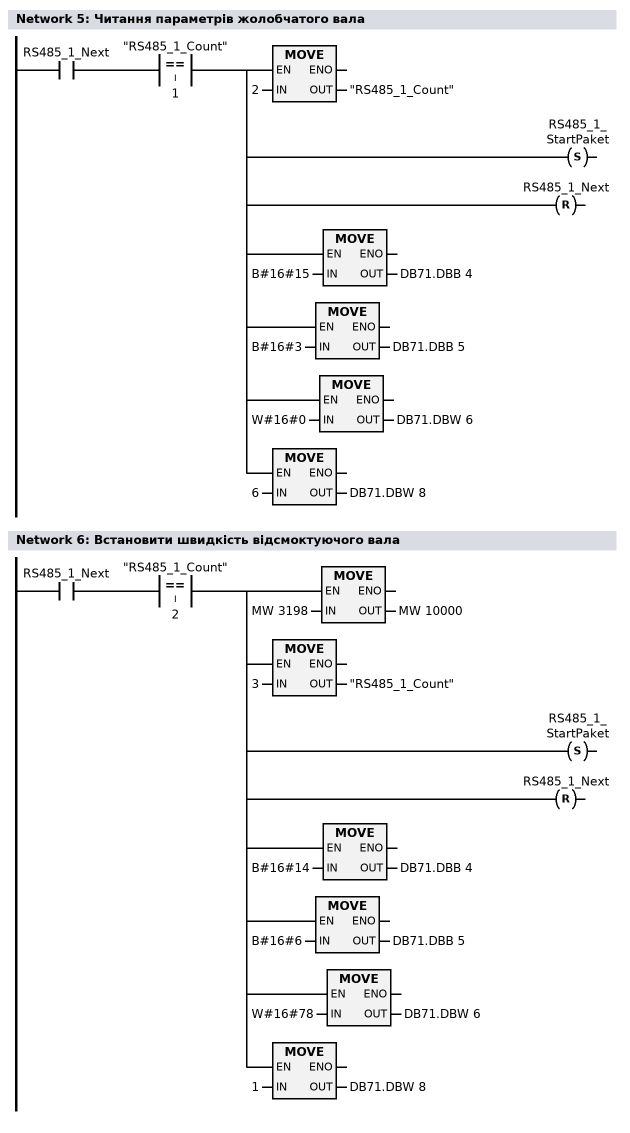
NETWORK
TITLE = Читання параметрів жолобчатого вала
      A     "RS485_1_Next";
      A(;
      L     "RS485_1_Count";
      L     1;
      ==I;
      );
      =     L 8.0;
      A     L 8.0;
      JNB   _007;
      L     2;
      T     "RS485_1_Count";
_007: NOP   0;
      A     L 8.0;
      BLD   102;
      S     "RS485_1_StartPaket";
      A     L 8.0;
      BLD   102;
      R     "RS485_1_Next";
      A     L 8.0;
      JNB   _008;
      L     B#16#15;
      T     DB71.DBB 4;
_008: NOP   0;
      A     L 8.0;
      JNB   _009;
      L     B#16#3;
      T     DB71.DBB 5;
_009: NOP   0;
      A     L 8.0;
      JNB   _00a;
      L     W#16#0;
      T     DB71.DBW 6;
_00a: NOP   0;
      A     L 8.0;
      JNB   _00b;
      L     6;
      T     DB71.DBW 8;
_00b: NOP   0;
NETWORK
TITLE = Встановити швидкість відсмоктуючого вала
      A     "RS485_1_Next";
      A(;
      L     "RS485_1_Count";
      L     2;
      ==I;
      );
      =     L 8.0;
      A     L 8.0;
      JNB   _00c;
      L     MW 3198;
      T     MW 10000;
_00c: NOP   0;
      A     L 8.0;
      JNB   _00d;
      L     3;
      T     "RS485_1_Count";
_00d: NOP   0;
      A     L 8.0;
      BLD   102;
      S     "RS485_1_StartPaket";
      A     L 8.0;
      BLD   102;
      R     "RS485_1_Next";
      A     L 8.0;
      JNB   _00e;
      L     B#16#14;
      T     DB71.DBB 4;
_00e: NOP   0;
      A     L 8.0;
      JNB   _00f;
      L     B#16#6;
      T     DB71.DBB 5;
_00f: NOP   0;
      A     L 8.0;
      JNB   _010;
      L     W#16#78;
      T     DB71.DBW 6;
_010: NOP   0;
      A     L 8.0;
      JNB   _011;
      L     1;
      T     DB71.DBW 8;
_011: NOP   0;
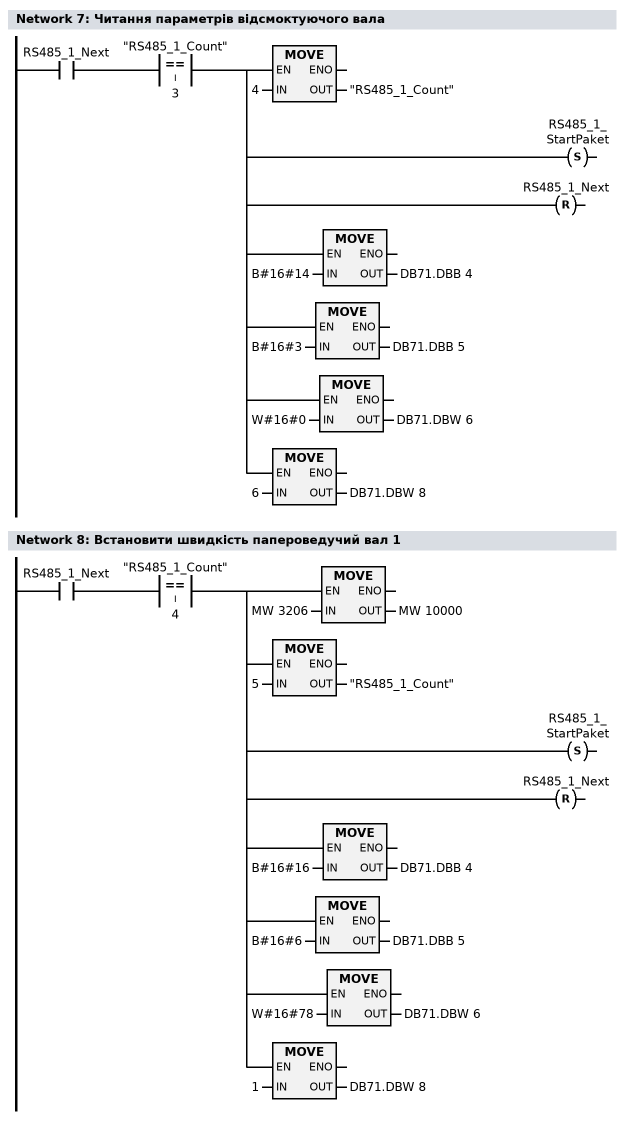
NETWORK
TITLE = Читання параметрів відсмоктуючого вала
      A     "RS485_1_Next";
      A(;
      L     "RS485_1_Count";
      L     3;
      ==I;
      );
      =     L 8.0;
      A     L 8.0;
      JNB   _012;
      L     4;
      T     "RS485_1_Count";
_012: NOP   0;
      A     L 8.0;
      BLD   102;
      S     "RS485_1_StartPaket";
      A     L 8.0;
      BLD   102;
      R     "RS485_1_Next";
      A     L 8.0;
      JNB   _013;
      L     B#16#14;
      T     DB71.DBB 4;
_013: NOP   0;
      A     L 8.0;
      JNB   _014;
      L     B#16#3;
      T     DB71.DBB 5;
_014: NOP   0;
      A     L 8.0;
      JNB   _015;
      L     W#16#0;
      T     DB71.DBW 6;
_015: NOP   0;
      A     L 8.0;
      JNB   _016;
      L     6;
      T     DB71.DBW 8;
_016: NOP   0;
NETWORK
TITLE = Встановити швидкість папероведучий вал 1
      A     "RS485_1_Next";
      A(;
      L     "RS485_1_Count";
      L     4;
      ==I;
      );
      =     L 8.0;
      A     L 8.0;
      JNB   _017;
      L     MW 3206;
      T     MW 10000;
_017: NOP   0;
      A     L 8.0;
      JNB   _018;
      L     5;
      T     "RS485_1_Count";
_018: NOP   0;
      A     L 8.0;
      BLD   102;
      S     "RS485_1_StartPaket";
      A     L 8.0;
      BLD   102;
      R     "RS485_1_Next";
      A     L 8.0;
      JNB   _019;
      L     B#16#16;
      T     DB71.DBB 4;
_019: NOP   0;
      A     L 8.0;
      JNB   _01a;
      L     B#16#6;
      T     DB71.DBB 5;
_01a: NOP   0;
      A     L 8.0;
      JNB   _01b;
      L     W#16#78;
      T     DB71.DBW 6;
_01b: NOP   0;
      A     L 8.0;
      JNB   _01c;
      L     1;
      T     DB71.DBW 8;
_01c: NOP   0;
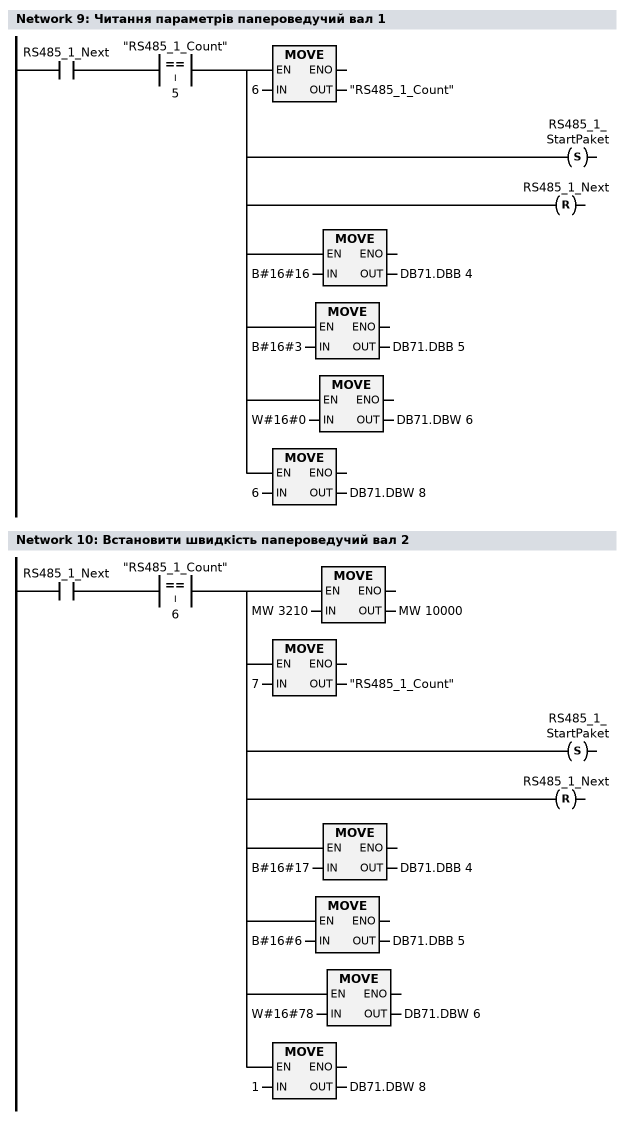
NETWORK
TITLE = Читання параметрів папероведучий вал 1
      A     "RS485_1_Next";
      A(;
      L     "RS485_1_Count";
      L     5;
      ==I;
      );
      =     L 8.0;
      A     L 8.0;
      JNB   _01d;
      L     6;
      T     "RS485_1_Count";
_01d: NOP   0;
      A     L 8.0;
      BLD   102;
      S     "RS485_1_StartPaket";
      A     L 8.0;
      BLD   102;
      R     "RS485_1_Next";
      A     L 8.0;
      JNB   _01e;
      L     B#16#16;
      T     DB71.DBB 4;
_01e: NOP   0;
      A     L 8.0;
      JNB   _01f;
      L     B#16#3;
      T     DB71.DBB 5;
_01f: NOP   0;
      A     L 8.0;
      JNB   _020;
      L     W#16#0;
      T     DB71.DBW 6;
_020: NOP   0;
      A     L 8.0;
      JNB   _021;
      L     6;
      T     DB71.DBW 8;
_021: NOP   0;
NETWORK
TITLE = Встановити швидкість папероведучий вал 2
      A     "RS485_1_Next";
      A(;
      L     "RS485_1_Count";
      L     6;
      ==I;
      );
      =     L 8.0;
      A     L 8.0;
      JNB   _022;
      L     MW 3210;
      T     MW 10000;
_022: NOP   0;
      A     L 8.0;
      JNB   _023;
      L     7;
      T     "RS485_1_Count";
_023: NOP   0;
      A     L 8.0;
      BLD   102;
      S     "RS485_1_StartPaket";
      A     L 8.0;
      BLD   102;
      R     "RS485_1_Next";
      A     L 8.0;
      JNB   _024;
      L     B#16#17;
      T     DB71.DBB 4;
_024: NOP   0;
      A     L 8.0;
      JNB   _025;
      L     B#16#6;
      T     DB71.DBB 5;
_025: NOP   0;
      A     L 8.0;
      JNB   _026;
      L     W#16#78;
      T     DB71.DBW 6;
_026: NOP   0;
      A     L 8.0;
      JNB   _027;
      L     1;
      T     DB71.DBW 8;
_027: NOP   0;
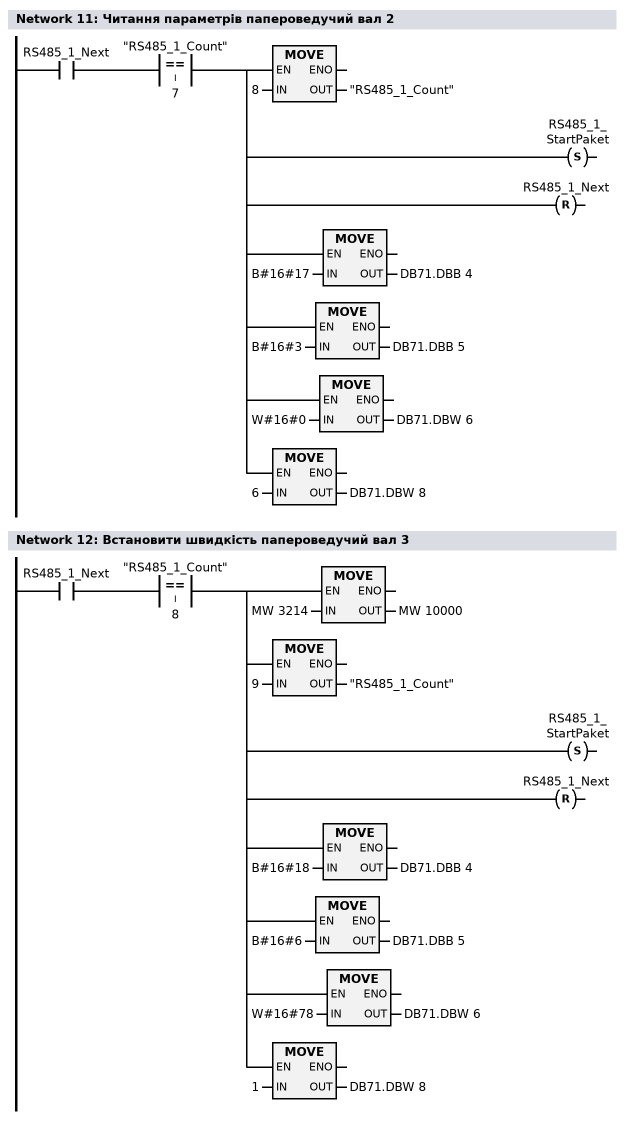
NETWORK
TITLE = Читання параметрів папероведучий вал 2
      A     "RS485_1_Next";
      A(;
      L     "RS485_1_Count";
      L     7;
      ==I;
      );
      =     L 8.0;
      A     L 8.0;
      JNB   _028;
      L     8;
      T     "RS485_1_Count";
_028: NOP   0;
      A     L 8.0;
      BLD   102;
      S     "RS485_1_StartPaket";
      A     L 8.0;
      BLD   102;
      R     "RS485_1_Next";
      A     L 8.0;
      JNB   _029;
      L     B#16#17;
      T     DB71.DBB 4;
_029: NOP   0;
      A     L 8.0;
      JNB   _02a;
      L     B#16#3;
      T     DB71.DBB 5;
_02a: NOP   0;
      A     L 8.0;
      JNB   _02b;
      L     W#16#0;
      T     DB71.DBW 6;
_02b: NOP   0;
      A     L 8.0;
      JNB   _02c;
      L     6;
      T     DB71.DBW 8;
_02c: NOP   0;
NETWORK
TITLE = Встановити швидкість папероведучий вал 3
      A     "RS485_1_Next";
      A(;
      L     "RS485_1_Count";
      L     8;
      ==I;
      );
      =     L 8.0;
      A     L 8.0;
      JNB   _02d;
      L     MW 3214;
      T     MW 10000;
_02d: NOP   0;
      A     L 8.0;
      JNB   _02e;
      L     9;
      T     "RS485_1_Count";
_02e: NOP   0;
      A     L 8.0;
      BLD   102;
      S     "RS485_1_StartPaket";
      A     L 8.0;
      BLD   102;
      R     "RS485_1_Next";
      A     L 8.0;
      JNB   _02f;
      L     B#16#18;
      T     DB71.DBB 4;
_02f: NOP   0;
      A     L 8.0;
      JNB   _030;
      L     B#16#6;
      T     DB71.DBB 5;
_030: NOP   0;
      A     L 8.0;
      JNB   _031;
      L     W#16#78;
      T     DB71.DBW 6;
_031: NOP   0;
      A     L 8.0;
      JNB   _032;
      L     1;
      T     DB71.DBW 8;
_032: NOP   0;
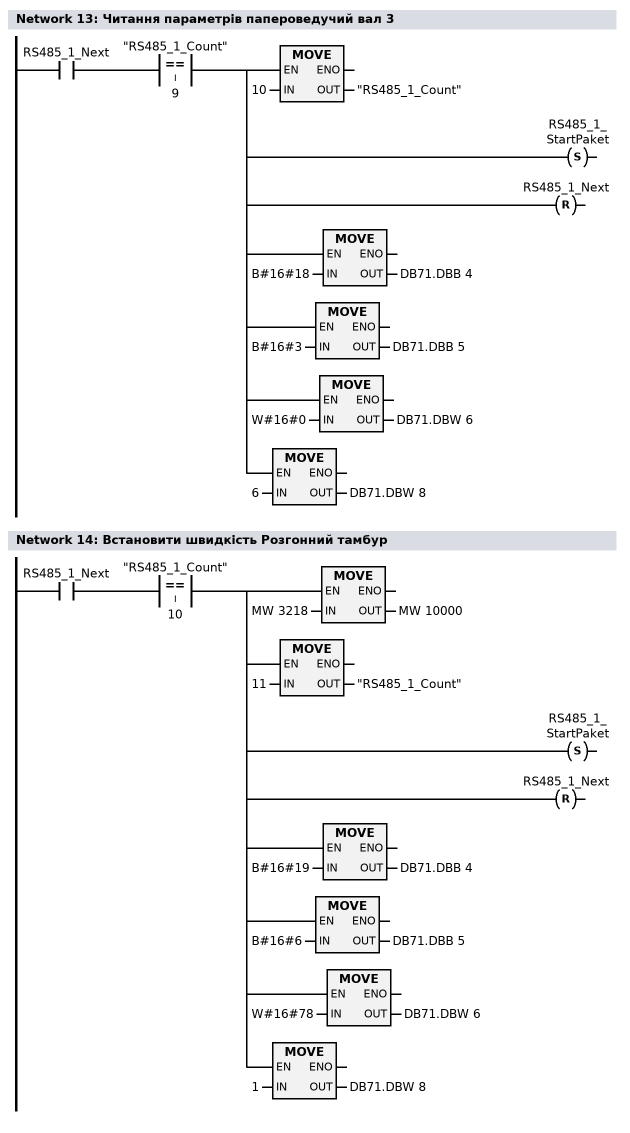
NETWORK
TITLE = Читання параметрів папероведучий вал 3
      A     "RS485_1_Next";
      A(;
      L     "RS485_1_Count";
      L     9;
      ==I;
      );
      =     L 8.0;
      A     L 8.0;
      JNB   _033;
      L     10;
      T     "RS485_1_Count";
_033: NOP   0;
      A     L 8.0;
      BLD   102;
      S     "RS485_1_StartPaket";
      A     L 8.0;
      BLD   102;
      R     "RS485_1_Next";
      A     L 8.0;
      JNB   _034;
      L     B#16#18;
      T     DB71.DBB 4;
_034: NOP   0;
      A     L 8.0;
      JNB   _035;
      L     B#16#3;
      T     DB71.DBB 5;
_035: NOP   0;
      A     L 8.0;
      JNB   _036;
      L     W#16#0;
      T     DB71.DBW 6;
_036: NOP   0;
      A     L 8.0;
      JNB   _037;
      L     6;
      T     DB71.DBW 8;
_037: NOP   0;
NETWORK
TITLE = Встановити швидкість Розгонний тамбур
      A     "RS485_1_Next";
      A(;
      L     "RS485_1_Count";
      L     10;
      ==I;
      );
      =     L 8.0;
      A     L 8.0;
      JNB   _038;
      L     MW 3218;
      T     MW 10000;
_038: NOP   0;
      A     L 8.0;
      JNB   _039;
      L     11;
      T     "RS485_1_Count";
_039: NOP   0;
      A     L 8.0;
      BLD   102;
      S     "RS485_1_StartPaket";
      A     L 8.0;
      BLD   102;
      R     "RS485_1_Next";
      A     L 8.0;
      JNB   _03a;
      L     B#16#19;
      T     DB71.DBB 4;
_03a: NOP   0;
      A     L 8.0;
      JNB   _03b;
      L     B#16#6;
      T     DB71.DBB 5;
_03b: NOP   0;
      A     L 8.0;
      JNB   _03c;
      L     W#16#78;
      T     DB71.DBW 6;
_03c: NOP   0;
      A     L 8.0;
      JNB   _03d;
      L     1;
      T     DB71.DBW 8;
_03d: NOP   0;
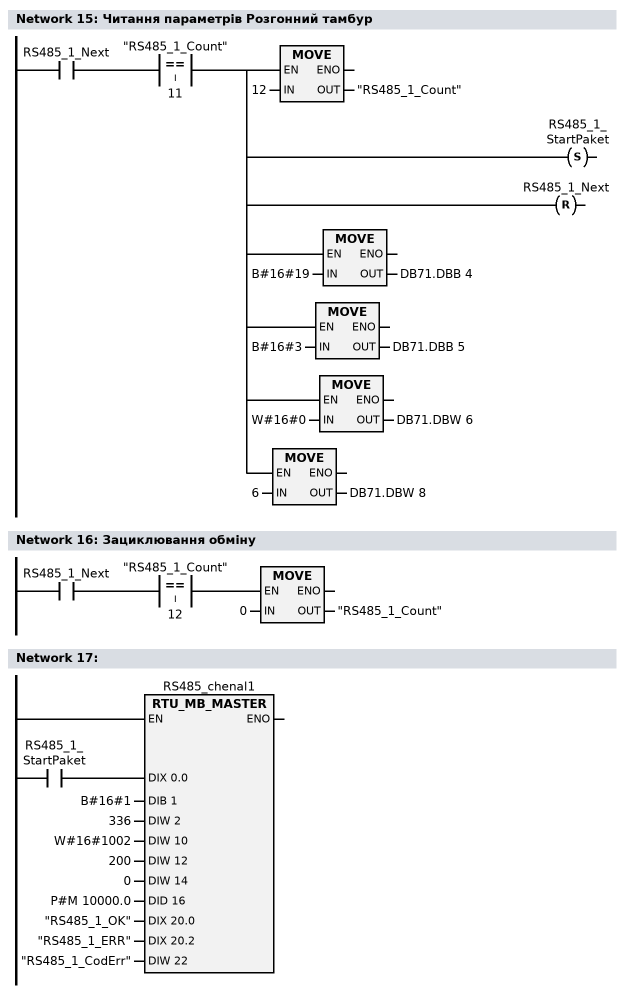
NETWORK
TITLE = Читання параметрів Розгонний тамбур
      A     "RS485_1_Next";
      A(;
      L     "RS485_1_Count";
      L     11;
      ==I;
      );
      =     L 8.0;
      A     L 8.0;
      JNB   _03e;
      L     12;
      T     "RS485_1_Count";
_03e: NOP   0;
      A     L 8.0;
      BLD   102;
      S     "RS485_1_StartPaket";
      A     L 8.0;
      BLD   102;
      R     "RS485_1_Next";
      A     L 8.0;
      JNB   _03f;
      L     B#16#19;
      T     DB71.DBB 4;
_03f: NOP   0;
      A     L 8.0;
      JNB   _040;
      L     B#16#3;
      T     DB71.DBB 5;
_040: NOP   0;
      A     L 8.0;
      JNB   _041;
      L     W#16#0;
      T     DB71.DBW 6;
_041: NOP   0;
      A     L 8.0;
      JNB   _042;
      L     6;
      T     DB71.DBW 8;
_042: NOP   0;
NETWORK
TITLE = Зациклювання обміну
      A     "RS485_1_Next";
      A(;
      L     "RS485_1_Count";
      L     12;
      ==I;
      );
      JNB   _043;
      L     0;
      T     "RS485_1_Count";
_043: NOP   0;
NETWORK
TITLE =
      A     "RS485_1_StartPaket";
      =     L 8.0;
      BLD   103;
      CALL  "RTU_MB_MASTER" , "RS485_chenal1" (
           DIX 0.0                  := L 8.0,
           DIB 1                    := B#16#1,
           DIW 2                    := 336,
           DIW 10                   := W#16#1002,
           DIW 12                   := 200,
           DIW 14                   := 0,
           DID 16                   := P#M 10000.0,
           DIX 20.0                 := "RS485_1_OK",
           DIX 20.2                 := "RS485_1_ERR",
           DIW 22                   := "RS485_1_CodErr");
      NOP   0;
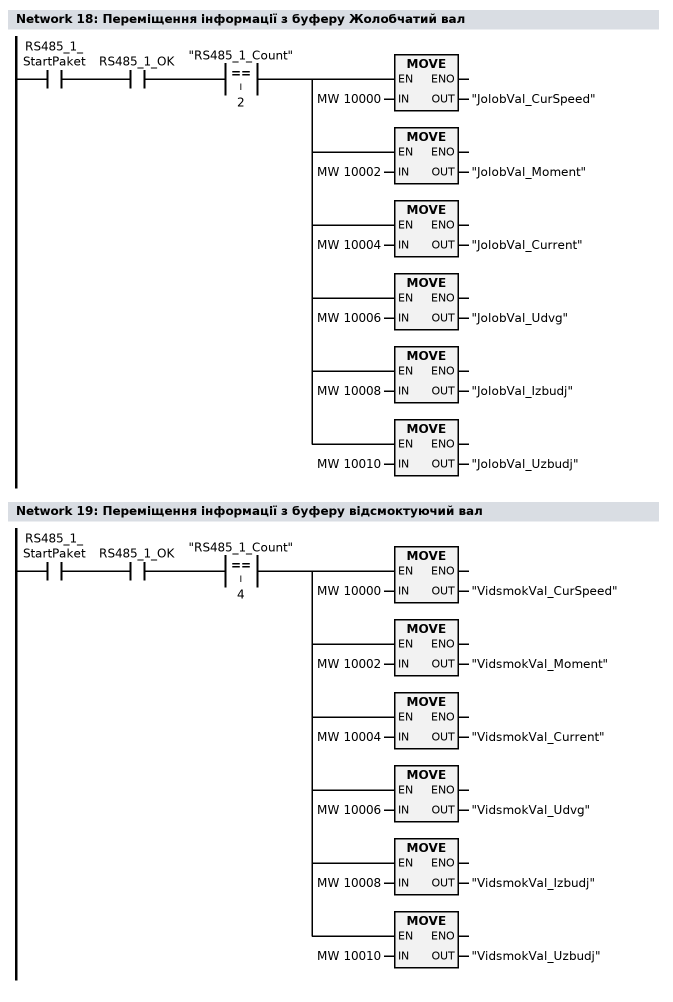
NETWORK
TITLE = Переміщення інформації з буферу Жолобчатий вал
      A     "RS485_1_StartPaket";
      A     "RS485_1_OK";
      A(;
      L     "RS485_1_Count";
      L     2;
      ==I;
      );
      =     L 8.0;
      A     L 8.0;
      JNB   _044;
      L     MW 10000;
      T     "JolobVal_CurSpeed";
_044: NOP   0;
      A     L 8.0;
      JNB   _045;
      L     MW 10002;
      T     "JolobVal_Moment";
_045: NOP   0;
      A     L 8.0;
      JNB   _046;
      L     MW 10004;
      T     "JolobVal_Current";
_046: NOP   0;
      A     L 8.0;
      JNB   _047;
      L     MW 10006;
      T     "JolobVal_Udvg";
_047: NOP   0;
      A     L 8.0;
      JNB   _048;
      L     MW 10008;
      T     "JolobVal_Izbudj";
_048: NOP   0;
      A     L 8.0;
      JNB   _049;
      L     MW 10010;
      T     "JolobVal_Uzbudj";
_049: NOP   0;
NETWORK
TITLE = Переміщення інформації з буферу відсмоктуючий вал
      A     "RS485_1_StartPaket";
      A     "RS485_1_OK";
      A(;
      L     "RS485_1_Count";
      L     4;
      ==I;
      );
      =     L 8.0;
      A     L 8.0;
      JNB   _04a;
      L     MW 10000;
      T     "VidsmokVal_CurSpeed";
_04a: NOP   0;
      A     L 8.0;
      JNB   _04b;
      L     MW 10002;
      T     "VidsmokVal_Moment";
_04b: NOP   0;
      A     L 8.0;
      JNB   _04c;
      L     MW 10004;
      T     "VidsmokVal_Current";
_04c: NOP   0;
      A     L 8.0;
      JNB   _04d;
      L     MW 10006;
      T     "VidsmokVal_Udvg";
_04d: NOP   0;
      A     L 8.0;
      JNB   _04e;
      L     MW 10008;
      T     "VidsmokVal_Izbudj";
_04e: NOP   0;
      A     L 8.0;
      JNB   _04f;
      L     MW 10010;
      T     "VidsmokVal_Uzbudj";
_04f: NOP   0;
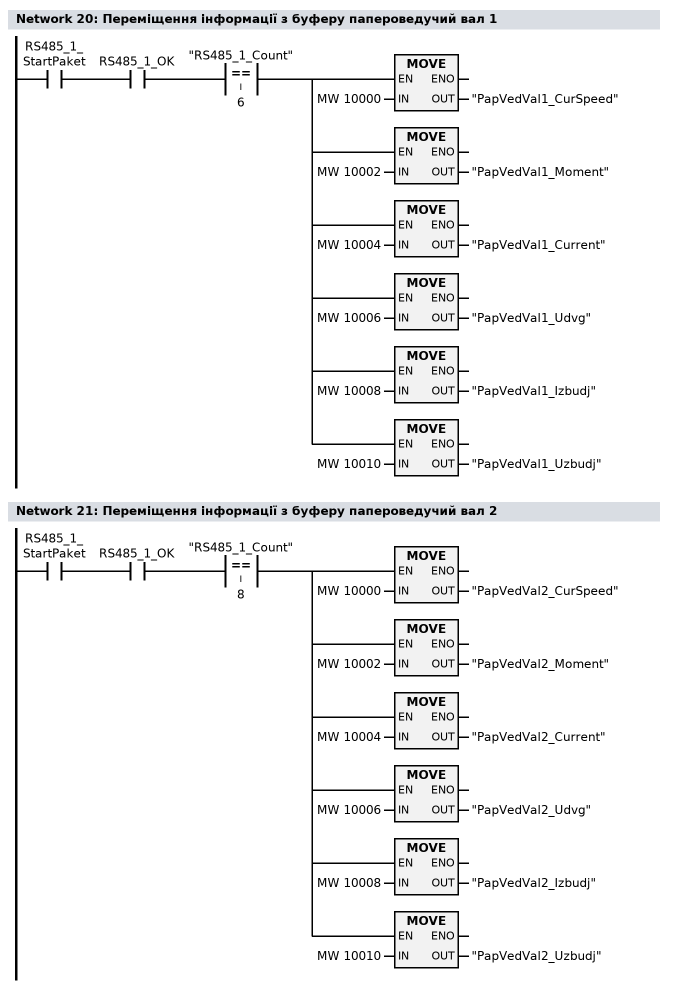
NETWORK
TITLE = Переміщення інформації з буферу папероведучий вал 1
      A     "RS485_1_StartPaket";
      A     "RS485_1_OK";
      A(;
      L     "RS485_1_Count";
      L     6;
      ==I;
      );
      =     L 8.0;
      A     L 8.0;
      JNB   _050;
      L     MW 10000;
      T     "PapVedVal1_CurSpeed";
_050: NOP   0;
      A     L 8.0;
      JNB   _051;
      L     MW 10002;
      T     "PapVedVal1_Moment";
_051: NOP   0;
      A     L 8.0;
      JNB   _052;
      L     MW 10004;
      T     "PapVedVal1_Current";
_052: NOP   0;
      A     L 8.0;
      JNB   _053;
      L     MW 10006;
      T     "PapVedVal1_Udvg";
_053: NOP   0;
      A     L 8.0;
      JNB   _054;
      L     MW 10008;
      T     "PapVedVal1_Izbudj";
_054: NOP   0;
      A     L 8.0;
      JNB   _055;
      L     MW 10010;
      T     "PapVedVal1_Uzbudj";
_055: NOP   0;
NETWORK
TITLE = Переміщення інформації з буферу папероведучий вал 2
      A     "RS485_1_StartPaket";
      A     "RS485_1_OK";
      A(;
      L     "RS485_1_Count";
      L     8;
      ==I;
      );
      =     L 8.0;
      A     L 8.0;
      JNB   _056;
      L     MW 10000;
      T     "PapVedVal2_CurSpeed";
_056: NOP   0;
      A     L 8.0;
      JNB   _057;
      L     MW 10002;
      T     "PapVedVal2_Moment";
_057: NOP   0;
      A     L 8.0;
      JNB   _058;
      L     MW 10004;
      T     "PapVedVal2_Current";
_058: NOP   0;
      A     L 8.0;
      JNB   _059;
      L     MW 10006;
      T     "PapVedVal2_Udvg";
_059: NOP   0;
      A     L 8.0;
      JNB   _05a;
      L     MW 10008;
      T     "PapVedVal2_Izbudj";
_05a: NOP   0;
      A     L 8.0;
      JNB   _05b;
      L     MW 10010;
      T     "PapVedVal2_Uzbudj";
_05b: NOP   0;
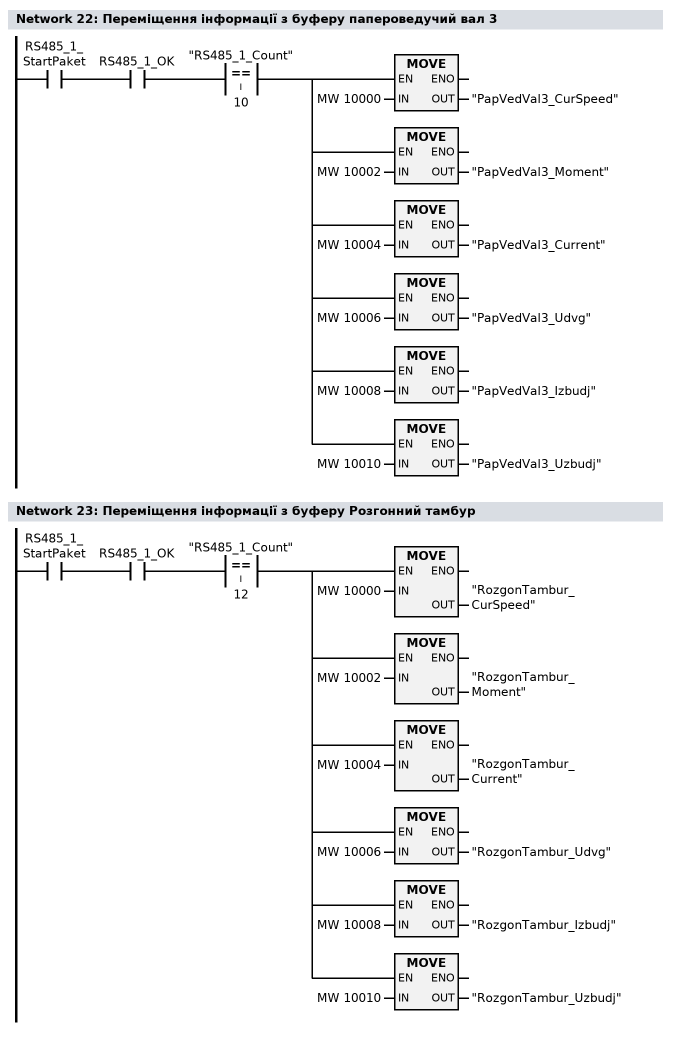
NETWORK
TITLE = Переміщення інформації з буферу папероведучий вал 3
      A     "RS485_1_StartPaket";
      A     "RS485_1_OK";
      A(;
      L     "RS485_1_Count";
      L     10;
      ==I;
      );
      =     L 8.0;
      A     L 8.0;
      JNB   _05c;
      L     MW 10000;
      T     "PapVedVal3_CurSpeed";
_05c: NOP   0;
      A     L 8.0;
      JNB   _05d;
      L     MW 10002;
      T     "PapVedVal3_Moment";
_05d: NOP   0;
      A     L 8.0;
      JNB   _05e;
      L     MW 10004;
      T     "PapVedVal3_Current";
_05e: NOP   0;
      A     L 8.0;
      JNB   _05f;
      L     MW 10006;
      T     "PapVedVal3_Udvg";
_05f: NOP   0;
      A     L 8.0;
      JNB   _060;
      L     MW 10008;
      T     "PapVedVal3_Izbudj";
_060: NOP   0;
      A     L 8.0;
      JNB   _061;
      L     MW 10010;
      T     "PapVedVal3_Uzbudj";
_061: NOP   0;
NETWORK
TITLE = Переміщення інформації з буферу Розгонний тамбур
      A     "RS485_1_StartPaket";
      A     "RS485_1_OK";
      A(;
      L     "RS485_1_Count";
      L     12;
      ==I;
      );
      =     L 8.0;
      A     L 8.0;
      JNB   _062;
      L     MW 10000;
      T     "RozgonTambur_CurSpeed";
_062: NOP   0;
      A     L 8.0;
      JNB   _063;
      L     MW 10002;
      T     "RozgonTambur_Moment";
_063: NOP   0;
      A     L 8.0;
      JNB   _064;
      L     MW 10004;
      T     "RozgonTambur_Current";
_064: NOP   0;
      A     L 8.0;
      JNB   _065;
      L     MW 10006;
      T     "RozgonTambur_Udvg";
_065: NOP   0;
      A     L 8.0;
      JNB   _066;
      L     MW 10008;
      T     "RozgonTambur_Izbudj";
_066: NOP   0;
      A     L 8.0;
      JNB   _067;
      L     MW 10010;
      T     "RozgonTambur_Uzbudj";
_067: NOP   0;
END_FUNCTION

